(* CoDeSys 2.3 library: beckhoff_network_112.lib *)
(* Libraries: oscat.lib 2.2.11 20:48:25, TcBase.lib 14.5.09 13:14:08, TcSystem.lib 9.3.10 12:21:30, TcpIp.lib 29.5.06 10:26:36, Standard.lib 5.6.98 13:03:02 *)

(* Global variable list: Constants *)
(* @OBJECTFLAGS := '0, 8' *)
VAR_GLOBAL CONSTANT
	NETWORK_BUFFER_LONG_SIZE : UINT := 3999;
	NETWORK_BUFFER_SHORT_SIZE : UINT := 1459;
	LOG_MAX : INT := 40;
	LOG_SIZE : INT := 80;
	ELEMENT_LENGTH : INT := 250;
END_VAR

(* Global variable list: Globale_Variablen *)
VAR_GLOBAL
	TCP_SERVER_RESET : BYTE; (* nur für TwinCAT notwendig ! *)
	LOG_CL : LOG_CONTROL;
END_VAR

(* Data type *)
TYPE DLOG_DATA :
STRUCT
	ADD_HEADER : BOOL;
	ADD_DATA : BOOL;
	CLOCK_TRIG : BOOL;
	ID_MAX : USINT;
	DTI : DT;
	UCB : UNI_CIRCULAR_BUFFER_DATA;
	NEW_FILE : STRING;
	NEW_FILE_RTRIG : BOOL;
END_STRUCT
END_TYPE

(* revision history
ks	01. oct. 2010	rev 1.0
	original version
*)

(* Data type *)
TYPE FILE_PATH_DATA :
STRUCT
	DRIVE : STRING(3);
	DIRECTORY : STRING(STRING_LENGTH);
	FILENAME : STRING;
END_STRUCT
END_TYPE

(* revision history
ks	01. oct. 2010	rev 1.0
	original version
*)

(* Data type *)
TYPE FILE_SERVER_DATA :
STRUCT
	FILE_OPEN : BOOL;
	FILENAME : STRING;
	MODE : BYTE;
	OFFSET : UDINT;
	FILE_SIZE : UDINT;
	AUTO_CLOSE : TIME;
	ERROR : BYTE;
END_STRUCT
END_TYPE

(* revision history
ks	01. oct. 2010	rev 1.0
	original version
*)

(* Data type *)
TYPE IP_C :
STRUCT
	C_MODE : BYTE;						(*W Mode: TCP/UCP AKTIV/PASSIV                               *)
	C_PORT : WORD;						(*W Portnummer                                               *)
	C_IP : DWORD;						(*W IP-Adresse gepackt wwxxyyzz = www.xxx.yyy.zzz            *)
	C_STATE : BYTE;						(*R Verbindungsstatus ON/OFF + Flanke ON/OFF                 *)
	C_ENABLE : BOOL;					(*W Freigabe für Connect                                     *)
	R_OBSERVE : BOOL;					(*W Empfang ueberwachen                                      *)
	TIME_RESET : BOOL;					(*W Alle Timer ruecksetzen                                   *)
	ERROR : DWORD;					(*R vvwwxxyy (vv = CON_ERROR, ww = SEN_ERROR, xx = REC_ERROR *)
	FIFO : IP_FIFO_DATA;					(*I IP FIFO Struktur                                         *)
	MAILBOX : ARRAY [1..16] OF BYTE;	(*I Mailbox: Datenbereich für Bausteindatenaustausch         *)
END_STRUCT
END_TYPE

(* revision history
ks	18. oct. 2008	rev 1.0
	original version
*)

(* Data type *)
TYPE IP_FIFO_DATA :
STRUCT
	X : ARRAY [1..128] OF BYTE; 	(* IP_ID FIFO Speicher          *)
	Y : ARRAY [1..128] OF BYTE; 	(* IP_ID Zähler                 *)
	ID : BYTE;					(* höchste vergabene id         *)
	MAX_ID : BYTE;				(* maximal Anmeldungen pro ID   *)
	INIT : BOOL;					(* Initialisierung durchgeführt *)
	EMPTY : BOOL;				(* FIFO leer                    *)
	FULL : BOOL;					(* FIFO voll                    *)
	TOP : INT;					(* maximale anzahl in FIFO      *)
	NW : INT;					(* Schreibzeiger                *)
	NR : INT;						(* Lesezeiger                   *)
END_STRUCT
END_TYPE

(* revision history
ks	18. oct. 2008	rev 1.0
	original version
*)

(* Data type *)
TYPE IP2GEO_DATA :
STRUCT
	STATE : BOOL;
	IP4 : DWORD;
	COUNTRY_CODE : STRING(2);
	COUNTRY_NAME : STRING(20);
	REGION_CODE : STRING(2);
	REGION_NAME : STRING(20);
	CITY : STRING(20);
	GEO_LATITUDE : REAL;
	GEO_LONGITUDE : REAL;
	TIME_ZONE_NAME : STRING(20);
	GMT_OFFSET : INT;
	IS_DST : BOOL;
END_STRUCT
END_TYPE

(* revision history
ks	14. aug. 2009	rev 1.0
	original version
*)

(* Data type *)
TYPE LOG_CONTROL :
STRUCT
	NEW_MSG : STRING(LOG_SIZE); (* neue Nachricht für den Datenbuffer *)
	NEW_MSG_OPTION : DWORD;
	LEVEL : BYTE;
	SIZE : INT := LOG_MAX; (* Anzahl der Strings im LOG_DATA *)
	RESET : BOOL; (* Nachrichtenbuffer löschen *)
	ENABLE : BOOL := TRUE; (* Debug Logging aktiv *)
	PRINTF : PRINTF_DATA; (* Array PRINTF Parameter *)
	MSG : ARRAY [0..LOG_MAX] OF STRING(LOG_SIZE); (* Array Message *)
	MSG_OPTION : ARRAY [0..LOG_MAX] OF DWORD; (* Array Options *)
	UPDATE_COUNT : UINT; (* Updatezähler *)
	IDX : INT; (* aktueller Nachrichten-Index *)
	RING_MODE : BOOL; (* Bufferüberlauf erkannt *)
END_STRUCT
END_TYPE

(* revision history
ks	18. oct. 2008	rev 1.0
	original version
*)

(* Data type *)
TYPE NETWORK_BUFFER :
STRUCT
	SIZE : UINT;
	BUFFER : NW_BUF_LONG;
END_STRUCT
END_TYPE

(* revision history
ks	01. 01. 2009	rev 1.0
	original version
*)

(* Data type *)
TYPE NETWORK_BUFFER_SHORT :
STRUCT
	SIZE : UINT;
	BUFFER : NW_BUF_SHORT;
END_STRUCT
END_TYPE

(* revision history
ks	01. 01. 2009	rev 1.0
	original version
*)

(* Data type *)
TYPE
	NW_BUF_LONG  : ARRAY[0..NETWORK_BUFFER_LONG_SIZE] OF BYTE;
END_TYPE

(* revision history
ks	01. 01. 2009	rev 1.0
	original version
*)

(* Data type *)
TYPE
	NW_BUF_SHORT : ARRAY[0..NETWORK_BUFFER_SHORT_SIZE] OF BYTE;
END_TYPE

(* revision history
ks	01. 01. 2009	rev 1.0
	original version
*)

(* Data type *)
TYPE PRINTF_DATA : ARRAY [1..11]  OF STRING(LOG_SIZE);
END_TYPE

(* revision history
ks	18. oct. 2008
	original version
*)

(* Data type *)
TYPE UNI_CIRCULAR_BUFFER_DATA :
STRUCT
	D_MODE : INT;
	D_HEAD : WORD;
	D_STRING : STRING(STRING_LENGTH);
	D_REAL : REAL;
	D_DWORD : DWORD;
	BUF_SIZE : UINT;
	BUF_COUNT : UINT;
	BUF_USED : USINT;
	BUF : NW_BUF_LONG;
	_GetStart : UINT;
	_GetEnd : UINT;
	_Last : UINT;
	_First : UINT;
END_STRUCT
END_TYPE

(* revision history
ks	01. oct. 2010	rev 1.0
	original version
*)

(* Data type *)
TYPE URL :
STRUCT
	PROTOCOL : STRING(10);
	USER : STRING(32);
	PASSWORD : STRING(32);
	DOMAIN : STRING(80);
	PORT : WORD;
	PATH : STRING(80);
	QUERY : STRING(STRING_LENGTH);
	ANCHOR : STRING(40);
	HEADER : STRING(160);
END_STRUCT
END_TYPE

(* revision history
hm	18. oct. 2008 v1.0
	original version

ks	01.oct.2010 v1.1
	new header element and string size
*)

(* Data type *)
TYPE us_LOG_VIEWPORT :
STRUCT
	LINE_ARRAY : ARRAY [1..40] OF INT;
	COUNT : INT; (* Anzahl der sichtbaren Nachtrichten *)
	UPDATE_COUNT : UINT; (* Updatezähler *)
	MOVE_TO_X : INT; (* Steuerung der Nachrichtenanzeige *)
	UPDATE : BOOL; (* Daten wurden geändert -> neuzeichnen *)
END_STRUCT
END_TYPE

(* revision history
ks	18. oct. 2008	rev 1.0
	original version
*)

(* Data type *)
TYPE us_TN_INPUT_CONTROL :
STRUCT
	bo_Enable: BOOL; (* Bearbeitung freigeben/sperren *)
	bo_Update_all: BOOL; (* All Elemente neu zeichnen *)
	bo_Reset_Fokus: BOOL; (* Fokus auf 1. Element setzen *)
	in_Focus_at: INT; (* Controlelement mit aktivem Fokus *)
	in_Count: INT; (* Anzahl der benutzen Control-Elemente *)
	in_ToolTip_X: INT; (* Tooltip Text X-Offset *)
	in_ToolTip_Y: INT; (* Tooltip Text Y-Offset *)
	by_ToolTip_Attr: BYTE; (* Tooltip Text Attribute *)
	in_ToolTip_Size: INT; (* Tooltip Text länge *)
	usa_TN_INPUT_CONTROL_DATA: ARRAY [1..20] OF us_TN_INPUT_CONTROL_DATA;
END_STRUCT
END_TYPE

(* revision history
ks	12. mai 2010	rev 1.0
	original version

*)

(* Data type *)
TYPE us_TN_INPUT_CONTROL_DATA :
STRUCT
 	by_Input_Exten_Code: BYTE;
	by_Input_ASCII_Code: BYTE;
	bo_Input_ASCII_IsNum: BOOL;
	in_Title_X_Offset: INT; (* Title Text X-Offset *)
	in_Title_Y_Offset: INT; (* Title Text Y-Offset *)
	by_Title_Attr: BYTE; (* Title Text Attribute *)
	st_Title_String: STRING; (* Title Text String *)
	in_Cursor_X: INT; (* aktuelle Cursor X-Position *)
	in_Cursor_Y: INT; (* aktuelle Cursor Y-Position *)
	in_Type: INT; (* Type des Elements *)
	in_X: INT; (* Element X-Position *)
	in_Y: INT; (* Element Y-Position *)
	in_Cursor_Pos: INT; (* aktuelle Cursorposition *)
	by_Attr_mF: BYTE; (* Text Attribute mit Fokus *)
	by_Attr_oF: BYTE; (* Text Attribute ohne Fokus *)
	in_selected: INT; (* Text Item wurde ausgewählt *)
	st_Input_Mask: STRING; (* Text Eingabemaske *)
	st_Input_Data: STRING(STRING_LENGTH); (* Text aktuelle Eingabedaten *)
	st_Input_String: STRING; (* Text Kopie nach Return-Taste *)
	st_Input_ToolTip: STRING; (* Text ToolTip (Eingabeinformation) *)
	in_Input_Option: INT; (* Text Ausgabe-Optionen *)
	bo_Input_Entered: BOOL; (* RETURN-Taste wurde betätigt *)
	bo_Input_Hidden: BOOL; (* Text versteckete Eingabe mit '*' *)
	bo_Input_Only_Num: BOOL; (* Text nur Nummerneingabe zulassen *)
	bo_Focus: BOOL; (* Element besitzt den Fokus *)
	bo_Update_Input: BOOL; (* Element wegen Benutzereingabe neuzeichnen *)
	bo_Update_All: BOOL; (* Element komplett neuzeichnen *)

END_STRUCT
END_TYPE

(* revision history
ks	12. mai 2010	rev 1.0
	original version

*)

(* Data type *)
TYPE us_TN_MENU :
STRUCT
	st_Menu_Text: STRING(STRING_LENGTH); (* X Menue Texte *)
	in_Menu_E_Count: INT; (* Menue Elemente Anzahl *)
	in_Y: INT; (* Menue Zeilennummer  Y-Position *)
	in_X: INT; (* Menue Spaltennummer X-Position *)
	by_Attr_mF: BYTE; (* Text Attribute mit Fokus *)
	by_Attr_oF: BYTE; (* Text Attribute ohne Fokus *)
	in_X_SM_new: INT; (* neue Sub-Menu X-Position *)
	in_Y_SM_new: INT; (* neue Sub-Menu Y-Position *)
	in_X_SM_old: INT; (* alte Sub-Menu X-Position *)
	in_Y_SM_old: INT; (* alte Sub-Menu Y-Position *)
	in_Cur_Menu_Item: INT; (* aktuelles Haupt-Menue *)
	in_Cur_Sub_Item: INT; (* aktuelles Sub-Menue *)
	in_State: INT; (*   Menu status   *)
	in_Menu_Selected: INT; (* X Menu-Item mit Enter angewwählt *)
	bo_Create: BOOL; (* X Menu erzeugen *)
	bo_Destroy: BOOL; (* X Menu entfernen *)
	bo_Update: BOOL; (* X Menu updaten *)
END_STRUCT
END_TYPE

(* revision history
ks	12. mai 2010	rev 1.0
	original version

*)

(* Data type *)
TYPE us_TN_MENU_POPUP :
STRUCT
	st_Menu_Text: STRING(STRING_LENGTH); (* X Menue Texte *)
	in_Menu_E_Count: INT; (* Menue Elemente Anzahl *)
	in_X: INT; (* X Menue X-Position *)
	in_Y: INT; (* X Menue Y-Position *)
	in_Cols: INT; (* Menue Spaltenanzahl *)
	in_Rows: INT; (* Menue Zeilenanzahl *)
	in_Cur_Item: INT; (* X aktuelles Sub-Menue *)
	by_Attr_mF: BYTE; (* X Text Attribute mit Fokus	*)
	by_Attr_oF: BYTE; (* X Text Attribute ohne Fokus *)
	by_Input_Exten_Code: BYTE; (* X Tastencode: Sondertasten *)
	bo_Create: BOOL; (* X Popup-Menu erzeugen *)
	bo_Destroy: BOOL; (* X Popup-Menu entfernen *)
	bo_Update: BOOL; (* X Popup-Menu updaten *)
	bo_Activ: BOOL; (*   Popup-Menu ist aktiv *)
END_STRUCT
END_TYPE

(* revision history
ks	12. mai 2010	rev 1.0
	original version

*)

(* Data type *)
TYPE us_TN_SCREEN :
STRUCT
	bya_CHAR: ARRAY [0..1919] OF BYTE;
	bya_COLOR: ARRAY [0..1919] OF BYTE;
	bya_BACKUP: ARRAY [0..1919] OF BYTE;
	bya_Line_Update: ARRAY [0..23] OF BOOL;
	by_Input_Exten_Code: BYTE;
	by_Input_ASCII_Code: BYTE;
	bo_Input_ASCII_IsNum: BOOL;
	in_Page_Number: INT; (* aktive Seiten-Nr. *)
	in_Cursor_X: INT; (* Cursor X-Position *)
	in_Cursor_Y: INT; (* Cursor Y-Position *)
	in_EOS_Offset: INT; (* End of String Offset *)
	by_Clear_Screen_Attr: BYTE; (* Clear-Screen Attr *)
	bo_Clear_Screen: BOOL; (* Clear-Screen auslösen *)
	bo_Modal_Dialog: BOOL; (* Modaler Dialog ist aktiv *)
	bo_Menue_Bar_Dialog: BOOL; (* Menue Dialog ist aktiv *)
END_STRUCT
END_TYPE

(* revision history
ks	12. mai 2010	rev 1.0
	original version

*)

(* Data type *)
TYPE VMAP_DATA :
STRUCT
	FC : DWORD;
	V_ADR : INT;
	V_SIZE : INT;
	P_ADR : INT;
	TIME_OUT : TIME;
END_STRUCT
END_TYPE

(* revision history
ks	18. oct. 2008	rev 1.0
	original version
*)

(* Data type *)
TYPE WORLD_WEATHER_CUR :
STRUCT
	OBSERVATION_TIME : STRING(8);
	TEMP_C : INT;
	WEATHER_CODE : INT;
	WEATHER_DESC : STRING(30);
	WIND_SPEED_MILES : INT;
	WIND_SPEED_KMPH : INT;
	WIND_DIR_DEGREE : INT;
	WIND_DIR16POINT : STRING(3);
	PRECIPMM : REAL;
	HUMIDITY : INT;
	VISIBILITY : INT;
	PRESSURE : INT;
	CLOUDOVER : INT;
END_STRUCT
END_TYPE

(* revision history
ks	01. oct. 2010	rev 1.0
	original version

*)

(* Data type *)
TYPE WORLD_WEATHER_DATA :
STRUCT
	CUR : WORLD_WEATHER_CUR;
	DAY : ARRAY [0..4] OF WORLD_WEATHER_DAY;
END_STRUCT
END_TYPE

(* revision history
ks	01. oct. 2010	rev 1.0
	original version

*)

(* Data type *)
TYPE WORLD_WEATHER_DAY :
STRUCT
	DATE_OF_DAY : STRING(10);
	TEMP_MAX_C : INT;
	TEMP_MAX_F : INT;
	TEMP_MIN_C : INT;
	TEMP_MIN_F : INT;
	WIND_SPEED_MILES : INT;
	WIND_SPEED_KMPH : INT;
	WIND_DIR_DEGREE : INT;
	WIND_DIR16POINT : STRING(3);
	WEATHER_CODE : INT;
	WEATHER_DESC : STRING(30);
	PRECIPMM : REAL;
END_STRUCT
END_TYPE

(* revision history
ks	01. oct. 2010	rev 1.0
	original version

*)

(* Data type *)
TYPE XML_CONTROL :
STRUCT
	COMMAND : WORD;
	WATCHDOG : TIME;
	START_POS : UINT;
	STOP_POS : UINT;
	COUNT : UINT;
	TYP : INT;
	LEVEL : UINT;
	PATH : STRING(STRING_LENGTH);
	ELEMENT : STRING(STRING_LENGTH);
	ATTRIBUTE : STRING(STRING_LENGTH);
	VALUE : STRING(STRING_LENGTH);
	BLOCK1_START : UINT;
	BLOCK1_STOP : UINT;
	BLOCK2_START : UINT;
	BLOCK2_STOP : UINT;
END_STRUCT
END_TYPE

(* revision history
ks	18. oct. 2008	rev 1.0
	original version

ks	24. sep. 2010	rev 1.1
	STRING(STRING_LENGTH)
*)

(* Data type *)
TYPE YAHOO_WEATHER_DATA :
STRUCT
	TIMETOLIVE : INT;							(* TIME TO LIVE: HOW LONG IN MINUTES THIS FEED SHOULD BE CACHED         *)
	LOCATION_CITY : STRING(40);   				(* THE LOCATION OF THIS FORECAST: CITY: CITY NAME  *)
	LOCATION_REGION : STRING(20);  				(* THE LOCATION OF THIS FORECAST: REGION: STATE, TERRITORY, OR REGION, IF GIVEN *)
	LOCATION_COUNTRY : STRING(20);			(* THE LOCATION OF THIS FORECAST: COUNTRY: TWO-CHARACTER COUNTRY CODE *)
	UNIT_TEMPERATURE : STRING(1);				(* TEMPERATURE: DEGREE UNITS, F FOR FAHRENHEIT OR C FOR CELSIUS *)
	UNIT_DISTANCE : STRING(2);					(* DISTANCE: UNITS FOR DISTANCE, MI FOR MILES OR KM FOR KILOMETERS *)
	UNIT_PRESSURE : STRING(2);					(* PRESSURE: UNITS OF BAROMETRIC PRESSURE, IN FOR POUNDS PER SQUARE INCH OR MB FOR MILLIBARS *)
	UNIT_SPEED : STRING(4);						(* SPEED: UNITS OF SPEED, MPH FOR MILES PER HOUR OR KPH FOR KILOMETERS PER HOUR *)
	WIND_CHILL : INT;							(* FORECAST INFORMATION ABOUT WIND CHILL IN DEGREES *)
	WIND_DIRECTION : INT;						(* FORECAST INFORMATION ABOUT WIND DIRECTION, IN DEGREES *)
	WIND_SPEED : REAL;							(* FORECAST INFORMATION ABOUT WIND SPEED, IN THE UNITS (MPH OR KPH)*)
	ATMOSPHERE_HUMIDITY : INT;				(* FORECAST INFORMATION ABOUT CURRENT ATMOSPHERIC HUMIDITY: HUMIDITY, IN PERCENT  *)
	ATMOSPHERE_PRESSURE : INT;				(* FORECAST INFORMATION ABOUT CURRENT ATMOSPHERIC PRESSURE: BAROMETRIC PRESSURE, IN THE UNITS (IN OR MB) *)
	ATMOSPHERE_VISIBILITY : REAL;				(* FORECAST INFORMATION ABOUT CURRENT ATMOSPHERIC VISIBILITY, IN THE UNITS (MI OR KM) *)
	ATMOSPHERE_RISING : INT;					(* FORECAST INFORMATION ABOUT RISING: STATE OF THE BAROMETRIC PRESSURE: STEADY (0), RISING (1), OR FALLING (2). (INTEGER: 0, 1, 2) *)
	ASTRONOMY_SUNRISE : STRING(10);			(* SUNRISE: TODAY'S SUNRISE TIME. THE TIME IS A STRING IN A LOCAL TIME FORMAT OF "H:MM AM/PM" *)
	ASTRONOMY_SUNSET : STRING(10);			(* SUNSET: TODAY'S SUNSET TIME. THE TIME IS A STRING IN A LOCAL TIME FORMAT OF "H:MM AM/PM", *)
	GEO_LATITUDE : REAL;						(* THE LATITUDE OF THE LOCATION *)
	GEO_LONGITUDE : REAL;						(* THE LONGITUDE OF THE LOCATION *)
	CUR_CONDITIONS_TEMP : INT;				(* THE CURRENT WEATHER CONDITIONS: TEMP: THE CURRENT TEMPERATURE, IN THE UNITS (F OR C) *)
	CUR_CONDITIONS_TEXT : STRING(40);			(* THE CURRENT WEATHER CONDITIONS: TEXT: A TEXTUAL DESCRIPTION OF CONDITIONS *)
	CUR_CONDITIONS_CODE : INT;				(* THE CURRENT WEATHER CONDITIONS: CODE: THE CONDITION CODE FOR THIS FORECAST *)
	FORCAST_TODAY_LOW_TEMP : INT;			(* THE FORCAST TODAY WEATHER CONDITIONS: THE FORECASTED LOW TEMPERATURE FOR THIS DAY IN THE UNITS (F OR C) *)
	FORCAST_TODAY_HIGH_TEMP : INT;			(* THE FORCAST TODAY WEATHER CONDITIONS: THE FORECASTED HIGH TEMPERATURE FOR THIS DAY IN THE UNITS (F OR C) *)
	FORCAST_TODAY_TEXT : STRING(40);			(* THE FORCAST TODAY WEATHER CONDITIONS: TEXT: A TEXTUAL DESCRIPTION OF CONDITIONS *)
	FORCAST_TODAY_CODE : INT;				(* THE CURRENT WEATHER CONDITIONS: CODE: THE CONDITION CODE FOR THIS FORECAST *)
	FORCAST_TOMORROW_LOW_TEMP : INT; 		(* THE FORCAST TOMORROW WEATHER CONDITIONS: THE FORECASTED LOW TEMPERATURE FOR THIS DAY IN THE UNITS (F OR C) *)
	FORCAST_TOMORROW_HIGH_TEMP : INT;		(* THE FORCAST TOMORROW WEATHER CONDITIONS: THE FORECASTED HIGH TEMPERATURE FOR THIS DAY IN THE UNITS (F OR C) *)
	FORCAST_TOMORROW_TEXT : STRING(40);	(* THE FORCAST TOMORROW WEATHER CONDITIONS: TEXT: A TEXTUAL DESCRIPTION OF CONDITIONS *)
	FORCAST_TOMORROW_CODE : INT;			(* THE CURRENT WEATHER CONDITIONS: CODE: THE CONDITION CODE FOR THIS FORECAST *)

END_STRUCT
END_TYPE

(* revision history
ks	18. oct. 2008	rev 1.0
	original version

ks	24. sep. 2010	rev 1.1
	LOCATION_COUNTRY STRING(20)

*)

(* POU BASE64_DEMO, CFC *)
PROGRAM BASE64_DEMO
VAR
	text1: STRING(144) := '<4036.1076324381@guildenstern.zeitform.de>';
	text2: STRING(192);
	text3: STRING(144);
	BASE64_DECODE_STR: BASE64_DECODE_STR;
	BASE64_ENCODE_STR: BASE64_ENCODE_STR;
	start: BOOL := TRUE;
	done1: BOOL;
	done2: BOOL;
END_VAR
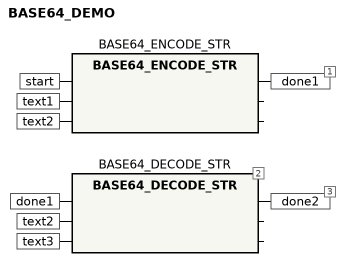
_CFC_ (* Continuous Function Chart, elements in execution order *)
#0 BASE64_ENCODE_STR:BASE64_ENCODE_STR(start, text1, text2)
#1 done1 <= #0.out 1
#2 BASE64_DECODE_STR:BASE64_DECODE_STR(done1, text2, text3)
#3 done2 <= #2.out 1
_END_CFC_
END_PROGRAM

(* POU BASE64_DECODE_STR, ST *)
FUNCTION_BLOCK BASE64_DECODE_STR
VAR_INPUT
	RUN : BOOL;
END_VAR
VAR_OUTPUT
	DONE : BOOL;
END_VAR
VAR_IN_OUT
	STR1 : STRING(192);
	STR2 : STRING(144);
END_VAR
VAR
	BASE64_DECODE_STREAM : BASE64_DECODE_STREAM;
	run_last : BOOL;
	buf1 : ARRAY [0..63] OF BYTE;
	buf2 : ARRAY [0..47] OF BYTE;
	mode : INT;
	size1 : INT;
	size2 : INT;
	end : INT;
	pos : INT;
END_VAR

(*
version 1.0	06. dec. 2009
programmer 	ks
tested by	ks

BASE64_DECODE_STR konvertiert einen BASE64 kodierten String in einen normalen String. 

*)
CASE mode OF
0:	IF RUN AND NOT run_last THEN
		DONE := FALSE;
		mode := 1;
		end := LEN(STR1);
		pos := 0;
		STR2 := '';
	END_IF;
1:
	size1 := MIN(48,end - pos);
	IF size1 > 0 THEN
		_STRING_TO_BUFFER(STR:=MID(STR1, size1, pos + 1), POS:=0, PT:=ADR(buf1), SIZE:=SIZEOF(buf1));
		BASE64_DECODE_STREAM(BUF1:=buf1 ,BUF2:=buf2 ,SIZE1:=size1 ,SIZE2=>size2);
		STR2 := CONCAT(STR2,BUFFER_TO_STRING(PT:=ADR(buf2), SIZE:=SIZEOF(buf2), START:=0, STOP:=size2 - 1));
	ELSE
		mode := 0;
		DONE := TRUE;
	END_IF;
	pos := pos + size1;
END_CASE;

run_last := RUN;

(* revision history

ks	6. dec. 2009 rev 1.0
	original version

*)
END_FUNCTION_BLOCK

(* POU BASE64_DECODE_STREAM, ST *)
FUNCTION_BLOCK BASE64_DECODE_STREAM
VAR_IN_OUT
	BUF1 : ARRAY [0..63] OF BYTE;
	BUF2 : ARRAY [0..47] OF BYTE;
END_VAR
VAR_INPUT
	SIZE1 : INT;
END_VAR
VAR_OUTPUT
	SIZE2 : INT;
END_VAR
VAR_TEMP
	a: INT;
	b: WORD;
	o: INT;
	off: INT;
	i1: INT;
	i2: INT;
	c: INT;
END_VAR

(*
version 1.0	06. dec. 2009
programmer 	ks
tested by	ks

BASE64_DECODE_STREAM konvertiert einzelne Base64 kodierte Datenblöcke in normalen Datenblöcke. 

*)
IF SIZE1 <= 0 THEN SIZE2 := 0; RETURN; END_IF;
c := SIZE1 - 1;
i2 := 0;
a := 0;
b := 0;
FOR i1 := 0 TO c DO
	o := BUF1[i1];
	IF o = 61  (* = *) THEN	EXIT;
	ELSIF o > 96 (* a-z *) THEN off := 71;
	ELSIF o > 64 (* A-Z *) THEN off := 65;
	ELSIF o > 47 (* 0-9 *) THEN off := -4;
	ELSIF o = 43 (* + *) THEN off := -19;
	ELSIF o = 47 (* / *) THEN off := -16;
	END_IF;
	b := SHL(b,6) OR INT_TO_BYTE(o - off);
	a := a + 6;
	IF a >= 8 THEN
		a := a - 8;
		BUF2[i2] := WORD_TO_BYTE(SHR(b,a));
		i2 := i2 + 1;
		b := b AND NOT SHL(WORD#16#FFFF,a);
	END_IF;
END_FOR;
SIZE2 := i2;

(* revision history

ks	6. dec. 2009 rev 1.0
	original version

*)
END_FUNCTION_BLOCK

(* POU BASE64_ENCODE_STR, ST *)
FUNCTION_BLOCK BASE64_ENCODE_STR
VAR_INPUT
	RUN : BOOL;
END_VAR
VAR_OUTPUT
	DONE : BOOL;
END_VAR
VAR_IN_OUT
	STR1 : STRING(144);
	STR2 : STRING(192);
END_VAR
VAR
	BASE64_ENCODE_STREAM : BASE64_ENCODE_STREAM;
	run_last : BOOL;
	buf1 : ARRAY [0..47] OF BYTE;
	buf2 : ARRAY [0..63] OF BYTE;
	mode : INT;
	size1 : INT;
	size2 : INT;
	end : INT;
	pos : INT;
END_VAR

(*
version 1.0	06. dec. 2009
programmer 	ks
tested by	ks

BASE64_ENCODE_STR konvertiert einen normalen String in einen BASE64 kodierten String. 

*)
CASE mode OF
0:	IF RUN AND NOT run_last THEN
		DONE := FALSE;
		mode := 1;
		end := LEN(STR1);
		pos := 0;
		STR2 := '';
	END_IF;
1:
	size1 := MIN(48,end - pos);
	IF size1 > 0 THEN
		_STRING_TO_BUFFER(STR:=MID(STR1, size1, pos + 1), POS:=0, PT:=ADR(buf1), SIZE:=SIZEOF(buf1));
		BASE64_ENCODE_STREAM(BUF1:=buf1 ,BUF2:=buf2 ,SIZE1:=size1 ,SIZE2=>size2);
		STR2 := CONCAT(STR2,BUFFER_TO_STRING(PT:=ADR(buf2), SIZE:=SIZEOF(buf2), START:=0, STOP:=size2 - 1));
	ELSE
		mode := 0;
		DONE := TRUE;
	END_IF;
	pos := pos + size1;
END_CASE;

run_last := RUN;

(* revision history

ks	6. dec. 2009 rev 1.0
	original version

*)
END_FUNCTION_BLOCK

(* POU BASE64_ENCODE_STREAM, ST *)
FUNCTION_BLOCK BASE64_ENCODE_STREAM
VAR_IN_OUT
	BUF1 : ARRAY [0..47] OF BYTE;
	BUF2 : ARRAY [0..63] OF BYTE;
END_VAR
VAR_INPUT
	SIZE1 : INT;
END_VAR
VAR_OUTPUT
	SIZE2 : INT;
END_VAR
VAR
	a: INT;
	b: WORD;
	i: INT;
	i2: INT;
	i3: INT;
	c: INT;
	BASE64: STRING(64) := 'ABCDEFGHIJKLMNOPQRSTUVWXYZabcdefghijklmnopqrstuvwxyz0123456789+/';
END_VAR

(*
version 1.0	06. dec. 2009
programmer 	ks
tested by	ks

BASE64_ENCODE_STREAM konvertiert Datenblöcke in Base64. 

*)
IF SIZE1 <= 0 THEN
	SIZE2 := 0;
	RETURN;
END_IF;
c := SIZE1 - 1;
i2 := 0;
a := 0;
b := 0;
FOR i := 0 TO c DO
	b := SHL(b,8) OR BUF1[i];
	a := a + 8;
	WHILE a >= 6 DO
		a := a - 6;
		buf2[i2] := CODE(BASE64,WORD_TO_INT(SHR(b,a)) + 1);
		i2 := i2 + 1;
		b := b AND NOT SHL(WORD#16#FFFF,a);
	END_WHILE;
END_FOR;
IF a > 0 THEN
	buf2[i2] := CODE(BASE64,WORD_TO_INT(SHL(b,6 - a)) + 1);
	i2 := i2 + 1;
	i3 := i2 + (NOT INT_TO_WORD(i2) AND 2#11);
	FOR i := i2 TO i3 DO
		buf2[i] := 61;
	END_FOR;
	SIZE2 := i3 + 1;
ELSE
	SIZE2 := i2;
END_IF;

(* revision history

ks	6. dec. 2009 rev 1.0
	original version

*)
END_FUNCTION_BLOCK

(* POU CSV_PARSER_BUF_DEMO, ST *)
PROGRAM CSV_PARSER_BUF_DEMO
VAR CONSTANT
	 line_cnt : INT:=2;
	 col_cnt : INT:=4;
END_VAR
VAR
	CPB : CSV_PARSER_BUF;
	FS : FILE_SERVER;
	FSD : FILE_SERVER_DATA;
	PT : NETWORK_BUFFER;
	sep : BYTE;
	value : STRING(STRING_LENGTH);
	step : INT;
	result : BYTE;
	offset : UDINT;
	run : BYTE;
	done : BOOL;
	value_real : REAL;
	cnt : INT;
	line : INT;
	idx : INT;
	data : ARRAY [1..line_cnt, 1..col_cnt] OF REAL;
	FB_LOG_MESSAGE : LOG_MSG;
END_VAR
(* Demo-Programm: CSV-Datei mittels Enumeration auswerten
die groesse des arrays kann mittels konstanten line_cnt und col_cnt angepasst werden

 ----- den nachfolgenden Textblock als datei "csv.txt" auf der sps ablegen ---
10.45,20,30,40.8
115,3450.2123,456,123.1
---------------------------------------------------------------------------------*)

CASE step OF

00:	IF NOT done THEN
	 	(* File_Daten einrichten  *)
		FSD.FILENAME := 'd:\pxc\oscat\network\csv.txt'; (* Dateiname *)
		FSD.MODE := 1; (* vorhandene Datei zum lesen öffnen *)
		FSD.OFFSET := 0; (* Start bei Dateianfang *)
		FSD.AUTO_CLOSE := T#0s; (* kein Auto-Close verwenden *)
		PT.SIZE := 65535; (* maximale länge einlesen *)
		step := 10;
	END_IF;

10:	IF FSD.MODE = 0 THEN (* Datei geöffnet ? *)
		OFFSET := 0; (* Start Offset vorgeben *)
		sep :=44; (* Trennzeichen , *)
		run := 1; (* Element suchen *)
		cnt := 0;
		step := 20;
	END_IF;

20:	IF run = 0 THEN
		(* ---------------------- Debug-Message ----------------------------*)
		IF LOG_CL.ENABLE THEN
			LOG_CL.NEW_MSG := 'CPFD: /value >~2< /offset ~3 /Run ~4 /Result ~5';
			LOG_CL.PRINTF[2] := value;
			LOG_CL.PRINTF[3] := UDINT_TO_STRING(OFFSET);
			LOG_CL.PRINTF[4] := BYTE_TO_STRING(run);
			LOG_CL.PRINTF[5] := BYTE_TO_STRING(result);
			FB_LOG_MESSAGE();
		END_IF;
		(* -----------------------------------------------------------------*)

		run := 1; (*  nächstes Element suchen  *)

		IF result = 1 OR result = 2 THEN
			(* automatische konvertierung in real ausführen *)
			IF LEN(value) <= 20 THEN
				value_real := FLOAT_TO_REAL(FLT:=value);
			ELSE
				value_real := 0.0;
			END_IF;

			cnt := cnt + 1;
			IF cnt <= line_cnt * col_cnt THEN
				line := (cnt / col_cnt) + 1;
				idx := (cnt MOD col_cnt);
				data[line,idx] := value_real; (* Daten in Array eintragen *)
			END_IF;

		ELSIF result = 10 THEN (* nichts mehr gefunden *)
			run := 0; (* keine weitere INI Auswertung erwünscht *)
			FSD.MODE := 5; (* Datei schliessen *)
			step := 30;
		END_IF;
	END_IF;

30:	IF FSD.MODE = 0 THEN (* Datei geschlossen ? *)
		step := 0;
		done := TRUE;
	END_IF;

END_CASE;

CPB(SEP:=sep,RUN:=run,OFFSET:=OFFSET,VALUE:=value,PT:=PT,RESULT=>result); (* CSV PARAMETER BUF *)
FS(FSD:=FSD,PT:=PT); (* FILE_SERVER *)
END_PROGRAM

(* POU CSV_PARSER_BUF, ST *)
FUNCTION_BLOCK CSV_PARSER_BUF
VAR_INPUT
	SEP : BYTE;
END_VAR
VAR_IN_OUT
	RUN : BYTE;
	OFFSET : UDINT;
	VALUE : STRING(STRING_LENGTH);
	PT : NETWORK_BUFFER;
END_VAR
VAR_OUTPUT
	RESULT : BYTE;
END_VAR
VAR
	step : INT;
	size : INT;
	c : BYTE;
	v_add : BYTE;
	i : INT;
	state : BYTE;
	eof : BOOL;
	pv : POINTER TO BYTE;
	pve : DWORD;
	watchdog : TON;
	x : BOOL;

	(*FB_LOG_MESSAGE : LOG_MSG;
	_debug_enable : BOOL := TRUE;
	step_last : INT;*)
END_VAR

(*
version 1.0		01. oct. 2010
programmer 		ks
tested by			ks

CSV_PARSER_BUF liefert die Elemente oder Zeilen einer Textdatei die in einem Bytearray abgelegt ist.

--------------------------------------

RUN Mode
00 = kein Befehl aktiv
01 = Element suchen

Result Codes
01 = Element gefunden
02 = Element und Zeilenende erkannt
05 = Befehl in Arbeit (Busy)
10 = nichts gefunden - Daten-Ende erreicht

State Codes
01 = Element gefunden
02 = Element und Zeilenende erkannt
05 = Befehl in Arbeit (Busy)
10 = nichts gefunden - Daten-Ende erreicht

*)
IF RUN > 0 THEN
	IF state = 0 THEN (* Auswertung neu beginnen *)

		pv := ADR(VALUE);
		pv^ := 0; (* VALUE = '' *)
		pve := pv + INT_TO_DWORD(STRING_LENGTH);
		i := UDINT_TO_INT(OFFSET);
		size := UINT_TO_INT(PT.SIZE) - 1;
		RESULT := 0;
		state := 5; (* Befehl in Arbeit (Busy) *)
		step := 0; (* Auswertung neu beginnen *)

		(* ---------------- Debug-Message -----------------------*)
		(*IF _debug_enable THEN
			LOG_CL.NEW_MSG := 'CPF: Startindex: ~1';
			LOG_CL.PRINTF[1] := INT_TO_STRING(i);
			FB_LOG_MESSAGE();
		END_IF;*)
		(* -----------------------------------------------------------------*)

	END_IF;

	watchdog(IN:=FALSE,PT:=T#1ms); (* Timer neustarten *)
	watchdog.IN := TRUE;

	WHILE (state = 5) DO (* Schleife solange kein Ergebnis *)

		watchdog(); (* Timer aktualisieren *)

		IF watchdog.Q THEN (* watchdog ausgelöst *)
			state := 5;
			EXIT;
		ELSIF i > size THEN (* kein weiteres zeichen vorhanden *)
			state := 10; (* nichts gefunden - Daten-Ende erreicht *)
			EXIT;
		ELSE

			c := PT.BUFFER[i]; (* neues Zeichen aus Buffer lesen *)
			eof := i + 1 = PT.SIZE; (* End of File *)

			v_add := 0;

			IF c = SEP THEN (* Neues Element erkannt *)
				state := 1;
				x := TRUE;
			ELSIF c >= 32 THEN (* Element erkannt *)
				v_add := c; (* Zeichen ablegen *)
				IF eof THEN
					state := 2; (* Element und Zeilenende erkannt *)
				ELSE
					x := TRUE;
				END_IF;
			ELSE
				IF x THEN
					state := 2; (* Element und Zeilenende erkannt *)
					x := FALSE;
				END_IF;
			END_IF;

			IF v_add > 0  AND pv < pve THEN (* Zeichen zu Value-String hinzufügen *)
				pv^ := v_add; (* Zeichen eintragen *)
				pv := pv + 1;
				pv^ := 0; (* String-Terminierung eintragen *)
			END_IF;

			i := i + 1; (* Datenzeiger erhöhen *)

		END_IF;
	END_WHILE;

	CASE state OF
	01:	(* Element gefunden *)
		RESULT := 1; (* Element gefunden *)
		OFFSET := i; (* Offset uebernehmen *)
		RUN := 0;
		state := 0;
	02:	(* Element gefunden *)
		RESULT := 2; (* Element und Zeilenende erkannt *)
		OFFSET := i; (* Offset uebernehmen *)
		RUN := 0;
		state := 0;

	05:	RESULT := 5; (* in Arbeit *)

	10:	(* Indexüberschreitung - Bufferende *)
		RESULT := 10; (* nichts gefunden - Datenende erreicht *)
		OFFSET := i; (* Offset uebernehmen *)
		RUN := 0;
		state := 0;
	END_CASE;

	(* ---------------- Debug-Message -----------------------*)
	(*IF _debug_enable THEN
		LOG_CL.NEW_MSG := 'CPF: intern Result ~1 , state ~2, step ~3 , offset ~4, run ~5';
		LOG_CL.PRINTF[1] := BYTE_TO_STRING(RESULT);
		LOG_CL.PRINTF[2] := BYTE_TO_STRING(state);
		LOG_CL.PRINTF[3] := INT_TO_STRING(step);
		LOG_CL.PRINTF[4] := UDINT_TO_STRING(OFFSET);
		LOG_CL.PRINTF[5] := BYTE_TO_STRING(RUN);
		FB_LOG_MESSAGE();
	END_IF;*)
	(* -----------------------------------------------------------------*)

END_IF;

(* ---------------- Debug-Message -----------------------*)
(*IF _debug_enable THEN
	IF step_last <> step THEN
		LOG_CL.NEW_MSG := 'IPB: Step: ~1';
		LOG_CL.PRINTF[1]  := INT_TO_STRING(step);
		FB_LOG_MESSAGE();
	END_IF;
	step_last := step;
END_IF;*)
(* -----------------------------------------------------------------*)

(* revision history
ks	01. oct. 2010	rev 1.0
	original version
*)
END_FUNCTION_BLOCK

(* POU FILE_SERVER, ST *)
FUNCTION_BLOCK FILE_SERVER
VAR_IN_OUT
	FSD : FILE_SERVER_DATA;
	PT : NETWORK_BUFFER;
END_VAR
VAR
	buf_size : UDINT;
	handle : UINT; (* Filehandle *)
	read_max_length : UDINT;(* maximale Datenlänge *)
	file_position : UDINT;(* aktueller Schreib/Lesezeiger *)
	used_filename : STRING;(* aktueller Dateiname *)
	close_time : TIME;
	length_read : UDINT;
	write_length : UDINT;
	length_written : UDINT;
	open_handle : UINT;
	seek_position : UDINT;
	seek_mode : INT;
	seek_data : ARRAY[0..1] OF DINT;
	tell_position : UDINT;
	open_mode : DWORD;
	last_mode: BYTE;
	command : BYTE;
	error_code : BYTE;
	error : BOOL;
	file_change : BOOL;
	step : INT;
	t_diff : TIME;
	tx_last : TIME;
	tx : TIME;
	X : FW_AdsRdWrt;
	tmpDW : UDINT;
	para : BOOL;

	(*FB_LOG_MESSAGE : LOG_MSG;
	_debug_enable : BOOL := TRUE;
	step_last : INT;*)
END_VAR

(*
version 1.0		23. sep. 2010
programmer 		ks
tested by			ks

FILE_SERVER ermöglicht den Zugriff auf Datteien mittels Plattform-Neutraler Schnittstelle
*)

(*
- Befehle -
1 = File_Open_Exist + File_Read
2 = File_Open_Exist + File_Write
3 = File_Open_New  + File_Write
4 = File_Remove
5 = File_Close

- Action -
1 = file_open (open)
2 = file_close (close)
3 = file_read (read)
4 = file_write (write)
5 = file_seek (setpos)
6 = file_tell (getpos)
7 = file_remove (delete)

---- fehlermeldungen----

00	Kein Fehler
19	SYSTEMSERVICE_FOPEN		Unbekannte oder ungültige Parameter
28	SYSTEMSERVICE_FOPEN		Datei nicht gefunden. Ungültiger Dateiname oder Dateipfad
38	SYSTEMSERVICE_FOPEN		Keine weiteren freien File Handles.
51	SYSTEMSERVICE_FCLOSE	ungültiges oder unbekanntes file handle.
62	SYSTEMSERVICE_FCLOSE	Datei wurde mit falscher Methode geöffnet.
67	SYSTEMSERVICE_FREAD		ungültiges oder unbekanntes file handle.
74	SYSTEMSERVICE_FREAD		Kein Speicher für Lesebuffer.
78	SYSTEMSERVICE_FREAD		Datei wurde mit falscher Methode geöffnet.
83	SYSTEMSERVICE_FWRITE	ungültiges oder unbekanntes file handle
94	SYSTEMSERVICE_FWRITE	Datei wurde mit falscher Methode geöffnet.
99	SYSTEMSERVICE_FSEEK		ungültiges oder unbekanntes file handle.
110	SYSTEMSERVICE_FSEEK		Datei wurde mit falscher Methode geöffnet.
115	SYSTEMSERVICE_FTELL		ungültiges oder unbekanntes file handle.
126	SYSTEMSERVICE_FTELL		Datei wurde mit falscher Methode geöffnet
140	SYSTEMSERVICE_FDELETE	Datei nicht gefunden. Ungültiger Dateiname oder Dateipfad.
255	Applikation					Position liegt hinter dem Dateiende

*)
(* read system timer *)
tx := UDINT_TO_TIME(T_PLC_MS());
t_diff := tx - tx_last;
tx_last := tx;

CASE step OF
0:
	IF FSD.MODE = LIMIT(1,FSD.MODE,5) THEN

		(* ---------------------- Debug-Message ----------------------------*)
		(*IF _debug_enable THEN
			LOG_CL.NEW_MSG := 'FS: File_Start Mode=~1';
			LOG_CL.PRINTF[1] := BYTE_TO_STRING(FSD.MODE);
			FB_LOG_MESSAGE();
		END_IF;*)
		(* -----------------------------------------------------------------------------*)

		(* Initialisierung *)
		X.sNetId := '';
		X.tTimeout := T#5s;
		X.nPort := 10000; (* AMSPORT_R3_SYSSERV *)

		buf_size := SIZEOF(PT.BUFFER);
		close_time := T#1ms; (* wenn Schritt aktiv ist, dann Close-Timer rücksetzen *)

		IF FSD.MODE = 4 THEN (* File_Remove *)
			IF handle > 0 THEN
				File_change := TRUE;
				step := 32000; (* File_Close ausführen *)
			ELSE
				step := 90; (* File_Remove ausführen *)
			END_IF;

		ELSIF FSD.MODE = 5 THEN (* File_Close *)
			step := 32000; (* File_Close ausführen *)

		ELSIF handle = 0 THEN (* MODE 1,2,3 *)
			step := 100; (* File muss erst geöffnet werden *)

		ELSE (* File ist geöffnset *)
			IF used_filename = FSD.FILENAME AND FSD.MODE = last_mode THEN (* kein Moduswechsel ? *)
				step := 200; (* ohne open prozedure weitermachen *)
			ELSE
				step := 32000;
				File_change := TRUE;
			END_IF;
		END_IF;

	ELSIF handle > 0 THEN (* offene Datei gefunden - AutoClose Modus *)
		IF FSD.AUTO_CLOSE > T#0s THEN
			close_time := close_time + t_diff; (* Close_Time hochzählen *)
			IF close_time > FSD.AUTO_CLOSE THEN (* Zeit überschrittenen *)
				step := 32000; (* automatisch Datei schliessen *)
			END_IF;
		END_IF;
	END_IF;

(* ----------------------------------- *)
090: (* File_Remove *)
	command := 7; (* File Remove *)
	step := 95;

095: (* File_Remove beendet *)
	IF command = 0 THEN
		step := 30000; (* Beenden *)
	END_IF;
(* ----------------------------------- *)

100: (* File_Open *)
	IF FSD.MODE = 3 THEN (* Open_New + File Write *)
		open_mode := 16#0001_001A; (* PATH_GENERIC + WRITEPLUS + BINARY *)
	ELSE (* Mode 1 Open_Exist + File _Read / Mode 2 Open_Exist + File_Write *)
		open_mode := 16#0001_0019; (* PATH_GENERIC + READPLUS + BINARY *)
	END_IF;
	command := 1; (* FileOpen *)
	step := 105;

105: (* File Open beendet *)
	IF command = 0 THEN
		IF error THEN
			step := 30000; (* Beenden *)
		ELSE
			(* Filedaten eintragen *)
			close_time := T#1ms; (* Timer freigeben *)
			handle := open_handle;
			used_filename := FSD.FILENAME;
			file_position := UDINT#4294967295; (* maximal = unbekannt *)
			last_mode := FSD.MODE;
			step := 110;
		END_IF;
	END_IF;

110: (* File Seek *)
	command := 5; (* File-Seek *)
	seek_position := 0;
	seek_mode := 2; (* SEEK_END - Seek from the end of file *)
	step := 115;

115: (* File Seek beendet *)
	IF command = 0 THEN
		IF error THEN
			step := 30000; (* Beenden *)
		ELSE
			command := 6; (* File-Tell starten *)
			step := 120;
		END_IF;
	END_IF;

120: (* File Tell beendet *)
	IF command = 0 THEN
		IF error THEN
			step := 30000; (* Beenden *)
		ELSE
			FSD.FILE_SIZE := tell_position; (* aktuelle Dateigroesse *)
			FSD.FILE_OPEN := TRUE;
			step := 200;
		END_IF;
	END_IF;

200: (* File Seek *)
	IF FSD.OFFSET > FSD.FILE_SIZE THEN (* prüfe auf gültige offset-vorgabe *)
		error_code := 255;
		step := 30000; (* Beenden *)
	ELSIF FSD.OFFSET <> file_position THEN
		command := 5; (* File-Seek *)
		seek_position := FSD.OFFSET;
		seek_mode := 0; (* Seek from beginning of file *)
		step := 210;
	ELSE
		step := 300;
	END_IF;

210: (* File Seek *)
	IF command = 0 THEN
		file_position := seek_position;
		IF error THEN
			step := 30000; (* Beenden *)
		ELSE
			step := 300;
		END_IF;
	END_IF;

300: (* Read or Write ? *)
	IF FSD.MODE = 1 THEN
		step := 400; (* Read *)
	ELSE
		step := 500; (* Write *)
	END_IF;

400: (* File Read *)
	IF UINT_TO_UDINT(PT.SIZE) > buf_size THEN (* Leselänge auf Buffergroesse begrenzen *)
		read_max_length := buf_size;
	ELSE
		read_max_length := UINT_TO_UDINT(PT.SIZE);
	END_IF;

	IF read_max_length > buf_size THEN
		read_max_length := buf_size;  (* Leselänge auf Buffergroesse begrenzen *)
	END_IF;

	(* Leselänge an Dateilänge anpassen *)
	IF file_position + read_max_length > FSD.FILE_SIZE THEN
		read_max_length := FSD.FILE_SIZE - file_position;
	END_IF;

	IF read_max_length > 0 THEN
		command := 3; (* File_Read *)
		step := 410;
	ELSE
		PT.SIZE := UINT#0;
		step := 30000; (* Beenden *)
	END_IF;

410: (* File Read *)
	IF command = 0 THEN
		PT.SIZE := UDINT_TO_UINT(length_read);
		IF NOT Error THEN
			file_position := file_position + length_read; (* aktueller File_Position korrigieren *)
			FSD.OFFSET := file_position;
		END_IF;
		step := 30000; (* Beenden *)
	END_IF;

500: (* File Write *)
	IF UINT_TO_UDINT(PT.SIZE) > buf_size THEN (* Schreiblänge auf Buffergroesse begrenzen *)
		write_length := buf_size;
	ELSE
		write_length := UINT_TO_UDINT(PT.SIZE);
	END_IF;

	IF write_length > 0 THEN
		command := 4; (* File_Write *)
		step := 510;
	ELSE
		step := 30000; (* Beenden *)
	END_IF;

510:
	IF command = 0 THEN
		IF NOT Error THEN
			file_position := file_position + length_written; (* aktueller File_Position korrigieren *)
			FSD.OFFSET := file_position;
			IF file_position > FSD.FILE_SIZE THEN (* Datei ist groesser geworden *)
				FSD.FILE_SIZE := file_position;
			END_IF;
		END_IF;
		step := 30000; (* Beenden *)
	END_IF;

 (* --------------------------------------------- *)

30000: (* Befehl fertig *)
	FSD.MODE := 0;
	FSD.ERROR := error_code;
	step := 0;

	(* ---------------- Debug-Message -----------------------*)
	(*IF _debug_enable THEN
		LOG_CL.NEW_MSG := 'FS: File_Stop: File ~1, error ~7, code ~8';
		LOG_CL.PRINTF[1]  := used_filename;
		LOG_CL.PRINTF[7]  := INT_TO_STRING(BOOL_TO_INT(error));
		LOG_CL.PRINTF[8]  := BYTE_TO_STRING(error_code);
		FB_LOG_MESSAGE();
	END_IF;*)
	(* --------------------------------------------- *)

32000:
	close_time := T#0s; (* Timer stoppen *)
	IF handle > 0 THEN
		command := 2; (* File_Close ausführen *)
	END_IF;
	step := 32100;

32100:
	IF command = 0 THEN (* File Close beendet *)
		(* Filedaten ablöschen *)
		FSD.FILE_OPEN := FALSE;
		file_position := 0;
		FSD.FILE_SIZE := 0;
		FSD.OFFSET := 0;
		used_filename := '';
		handle := 0;

		(* File_Name wurde fliegend geändert ? *)
		IF file_change THEN
			file_change := FALSE;
			step := 0;
		ELSE
			step := 30000;
		END_IF;
	END_IF;

END_CASE;

(* 1 = file_open
   2 = file_close
   3 = file_read
   4 = file_write
   5 = file_seek
   6 = file_tell
   7 = file_remove
*) 

X(bExecute := FALSE); (* Zyklischer FW_AdsRdWrt Aufruf *)

(* ------------ File Open ------------- *)
IF command = 1 THEN
	IF NOT para THEN
		para := TRUE;
		X(	nIdxGrp := 120, (* SYSTEMSERVICE_FOPEN *)
			nidxOffs := open_mode,
			cbWriteLen := SIZEOF(FSD.FILENAME),
			pWriteBuff := ADR(FSD.FILENAME),
			cbReadLen := SIZEOF(tmpDW),
			pReadBuff := ADR(tmpDW),
			bExecute := TRUE
			);
	ELSIF X.bBusy = FALSE THEN
		para := FALSE;
		error := X.bError;
		error_code := SEL(error,0,UDINT_TO_BYTE(X.nErrId + 16#10));

		IF X.cbRead >= SIZEOF(tmpDW) THEN
			open_handle := UDINT_TO_UINT(tmpDW);
		ELSE
			open_handle := 0;
		END_IF;
		command := 0;

		(* ---------------- Debug-Message -----------------------*)
		(*IF _debug_enable THEN
			LOG_CL.NEW_MSG := 'FS: Open: File ~1, handle ~2 , mode ~3 , error ~7, code ~8';
			LOG_CL.PRINTF[1] := FSD.FILENAME;
			LOG_CL.PRINTF[2] := DWORD_TO_STRING(open_handle);
			LOG_CL.PRINTF[3] := DWORD_TO_STRING(open_mode);
			LOG_CL.PRINTF[7] := INT_TO_STRING(BOOL_TO_INT(error));
			LOG_CL.PRINTF[8] := BYTE_TO_STRING(error_code);
			FB_LOG_MESSAGE();
		END_IF;*)
		(* -----------------------------------------------------------------*)
	END_IF;
END_IF;

(* ----------- File Close ------------- *)
IF command = 2 THEN
	IF NOT para THEN
		para := TRUE;
		X(	nIdxGrp := 121, (* SYSTEMSERVICE_FCLOSE *)
			nidxOffs := handle,
			cbWriteLen := 0,
			pWriteBuff := 0,
			cbReadLen := 0,
			pReadBuff := 0,
			bExecute := TRUE
			);
	ELSIF X.bBusy = FALSE THEN
		para := FALSE;
		error := X.bError;
		error_code := SEL(error,0,UDINT_TO_BYTE(X.nErrId + 16#30));
		command := 0;
		(* ---------------- Debug-Message -----------------------*)
		(*IF _debug_enable THEN
			LOG_CL.NEW_MSG := 'FS: Close: File ~1, error ~7, code ~8';
			LOG_CL.PRINTF[1] := used_filename;
			LOG_CL.PRINTF[7] := INT_TO_STRING(BOOL_TO_INT(error));
			LOG_CL.PRINTF[8] := BYTE_TO_STRING(error_code);
			FB_LOG_MESSAGE();
		END_IF;*)
		(* -----------------------------------------------------------------*)
	END_IF;
END_IF;

(* ------------ File Read ------------- *)
IF command = 3 THEN
	IF NOT para THEN
		para := TRUE;
		X(	nIdxGrp := 122, (* SYSTEMSERVICE_FREAD *)
			nidxOffs := handle,
			cbWriteLen := 0,
			pWriteBuff := 0,
			cbReadLen := read_max_length,
			pReadBuff := ADR(PT.BUFFER),
			bExecute := TRUE
			);
	ELSIF X.bBusy = FALSE THEN
		length_read := X.cbRead;
		para := FALSE;
		error := X.bError;
		error_code := SEL(error,0,UDINT_TO_BYTE(X.nErrId + 16#40));
		command := 0;

		(* ---------------- Debug-Message -----------------------*)
		(*IF _debug_enable THEN
			LOG_CL.NEW_MSG := 'FS: Read: File ~1, soll ~2,ist ~3 ,error ~7, code ~8';
			LOG_CL.PRINTF[1] := used_filename;
			LOG_CL.PRINTF[2] := UDINT_TO_STRING(read_max_length);
			LOG_CL.PRINTF[3] := UDINT_TO_STRING(length_read);
			LOG_CL.PRINTF[7] := INT_TO_STRING(BOOL_TO_INT(error));
			LOG_CL.PRINTF[8] := BYTE_TO_STRING(error_code);
			FB_LOG_MESSAGE();
		END_IF;*)
		(* -----------------------------------------------------------------*)
	END_IF;
END_IF;

(* ------------ File Write ------------- *)
IF command = 4 THEN
	IF NOT para THEN
		para := TRUE;
		X(	nIdxGrp := 123, (* SYSTEMSERVICE_FWRITE *)
			nidxOffs := handle,
			cbWriteLen := write_length,
			pWriteBuff := ADR(PT.BUFFER),
			cbReadLen := SIZEOF(length_written),
			pReadBuff := ADR(length_written),
			bExecute := TRUE
			);
	ELSIF X.bBusy = FALSE THEN
		para := FALSE;
		error := X.bError;
		error_code := SEL(error,0,UDINT_TO_BYTE(X.nErrId + 16#50));
		command := 0;

		(* ---------------- Debug-Message -----------------------*)
		(*IF _debug_enable THEN
			LOG_CL.NEW_MSG := 'FS: Write: File ~1, soll ~2,ist ~3 ,error ~7, code ~8';
			LOG_CL.PRINTF[1] := used_filename;
			LOG_CL.PRINTF[2] := UDINT_TO_STRING(write_length);
			LOG_CL.PRINTF[3] := UDINT_TO_STRING(length_written);
			LOG_CL.PRINTF[7] := INT_TO_STRING(BOOL_TO_INT(error));
			LOG_CL.PRINTF[8] := BYTE_TO_STRING(error_code);
			FB_LOG_MESSAGE();
		END_IF;*)
		(* -----------------------------------------------------------------*)
	END_IF;
END_IF;

(* ------------ File Seek ------------- *)
IF command = 5 THEN
	IF NOT para THEN
		para := TRUE;
		seek_data[0] := UDINT_TO_DINT(seek_position);
		seek_data[1] := INT_TO_DINT(seek_mode);

		X(	nIdxGrp := 124, (* SYSTEMSERVICE_FSEEK *)
			nidxOffs := handle,
			cbWriteLen := SIZEOF(seek_data),
			pWriteBuff := ADR(seek_data),
			cbReadLen := 0,
			pReadBuff := 0,
			bExecute := TRUE
			);
	ELSIF X.bBusy = FALSE THEN
		para := FALSE;
		error := X.bError;
		error_code := SEL(error,0,UDINT_TO_BYTE(X.nErrId + 16#60));
		command := 0;

		(* ---------------- Debug-Message -----------------------*)
		(*IF _debug_enable THEN
			LOG_CL.NEW_MSG := 'FS: Seek: File ~1,pos ~3 ,error ~7, code ~8';
			LOG_CL.PRINTF[1] := used_filename;
			LOG_CL.PRINTF[3] := UDINT_TO_STRING(seek_position);
			LOG_CL.PRINTF[7] := INT_TO_STRING(BOOL_TO_INT(error));
			LOG_CL.PRINTF[8] := BYTE_TO_STRING(error_code);
			FB_LOG_MESSAGE();
		END_IF;*)
		(* -----------------------------------------------------------------*)
	END_IF;
END_IF;

(* ------------ File Tell ------------- *)
IF command = 6 THEN
	IF NOT para THEN
		para := TRUE;
		X(	nIdxGrp := 125, (* SYSTEMSERVICE_FTELL *)
			nidxOffs := handle,
			cbWriteLen := 0,
			pWriteBuff := 0,
			cbReadLen := SIZEOF(tell_position),
			pReadBuff := ADR(tell_position),
			bExecute := TRUE
			);
	ELSIF X.bBusy = FALSE THEN
		para := FALSE;
		error := X.bError;
		error_code := SEL(error,0,UDINT_TO_BYTE(X.nErrId + 16#70));
		command := 0;

		(* ---------------- Debug-Message -----------------------*)
		(*IF _debug_enable THEN
			LOG_CL.NEW_MSG := 'FS: Tell: File ~1, pos ~3 ,error ~7, code ~8';
			LOG_CL.PRINTF[1] := used_filename;
			LOG_CL.PRINTF[3] := UDINT_TO_STRING(tell_position);
			LOG_CL.PRINTF[7] := INT_TO_STRING(BOOL_TO_INT(error));
			LOG_CL.PRINTF[8] := BYTE_TO_STRING(error_code);
			FB_LOG_MESSAGE();
		END_IF;*)
		(* -----------------------------------------------------------------*)
	END_IF;
END_IF;

(* ------------ File Remove ------------- *)
IF command = 7 THEN
	IF NOT para THEN
		para := TRUE;
		X(	nIdxGrp := 131, (* SYSTEMSERVICE_FDELETE *)
			nidxOffs := 16#0001_0000, (* PATH_GENERIC *)
			cbWriteLen := SIZEOF(FSD.FILENAME),
			pWriteBuff := ADR(FSD.FILENAME),
			cbReadLen := 0,
			pReadBuff := 0,
			bExecute := TRUE
			);
	ELSIF X.bBusy = FALSE THEN
		para := FALSE;
		error := X.bError;
		error_code := SEL(error,0,UDINT_TO_BYTE(X.nErrId + 16#80));
		command := 0;

		(* ---------------- Debug-Message -----------------------*)
		(*IF _debug_enable THEN
			LOG_CL.NEW_MSG := 'FS: Remove: File ~1, error ~7, code ~8';
			LOG_CL.PRINTF[1] := FSD.FILENAME;
			LOG_CL.PRINTF[7] := INT_TO_STRING(BOOL_TO_INT(error));
			LOG_CL.PRINTF[8] := BYTE_TO_STRING(error_code);
			FB_LOG_MESSAGE();
		END_IF;*)
		(* -----------------------------------------------------------------*)
	END_IF;
END_IF;

(* ---------------- Debug-Message -----------------------*)
(*IF _debug_enable THEN
	IF step_last <> step THEN
		LOG_CL.NEW_MSG := 'FS: Step: ~1';
		LOG_CL.PRINTF[1] := INT_TO_STRING(step);
		FB_LOG_MESSAGE();
	END_IF;
	step_last := step;
END_IF;*)
(* -----------------------------------------------------------------*)

(* revision history
ks	23. sep. 2010	rev 1.0
	original version
*)
END_FUNCTION_BLOCK

(* POU LOG_MSG, ST *)
FUNCTION_BLOCK LOG_MSG
(* VAR_EXTERNAL
	LOG_CL :	LOG_CONTROL;
END_VAR *)
VAR
	FB_PRINT_SF :PRINT_SF;
	idX : INT;
END_VAR

(*
version 1.0		01 mai 2010
programmer		ks
tested by		ks

LOG_MSG trägt Meldungen in den Loggingbuffer ein
*)
IF DWORD_TO_BYTE(SHL(LOG_CL.NEW_MSG_OPTION,16)) > LOG_CL.LEVEL OR NOT LOG_CL.ENABLE THEN RETURN; END_IF; (* Logging freigegeben ?*)

FB_PRINT_SF(PRINTF_DATA := LOG_CL.PRINTF,STR := LOG_CL.NEW_MSG);

IF LOG_CL.RESET THEN (* Logeinträge löschen *)
	LOG_CL.RESET := FALSE;
	LOG_CL.RING_MODE := FALSE;
	LOG_CL.IDX := 0;
	LOG_CL.UPDATE_COUNT := LOG_CL.UPDATE_COUNT + UINT#1; (* UpdateCount erhöhen *)
END_IF;

IF LOG_CL.SIZE > 0 THEN (* size wert ist eingetragen *)
	IF LEN(LOG_CL.NEW_MSG) > 0 THEN (* Meldung in Puffer eintragen *)
		IF (LOG_CL.IDX >= LOG_CL.SIZE) THEN
			LOG_CL.RING_MODE := TRUE; (* bei Überlauf = Ringbuffermodus *)
			LOG_CL.IDX := 0; (* wieder auf arrayanfang positionieren *)
		END_IF;

		LOG_CL.UPDATE_COUNT := LOG_CL.UPDATE_COUNT + UINT#1; (* UpdateCount erhöhen *)
		LOG_CL.IDX := LOG_CL.IDX + INT#1; (* nächste freie Position *)
		idx := LOG_CL.IDX; (* lade aktuelle Log-Puffer Positition *)
		LOG_CL.MSG[idx] := LOG_CL.NEW_MSG; (* neuen Log-String in puffer ablegen  *)
		LOG_CL.MSG_OPTION[idx] := LOG_CL.NEW_MSG_OPTION; (* neue Log-String Option in puffer ablegen  *)
		LOG_CL.NEW_MSG := ''; (* letzten Log-String löschen *)
	END_IF;
END_IF;
END_FUNCTION_BLOCK

(* POU PRINT_SF, ST *)
FUNCTION_BLOCK PRINT_SF
VAR_IN_OUT
	PRINTF_DATA : PRINTF_DATA;
	STR : STRING(LOG_SIZE);
END_VAR
VAR
	pos : INT;
	c : INT;
	src : STRING(1) := '~';
	run : BOOL;
END_VAR

(*

version 1.0 		14. aug. 2009
programmer 	ks
tested by		ks

PRINTF erzeugt aus einem Parameterstring und den übergebenen Parameterdaten einen Text
*)
IF LEN(STR) > 0 THEN
	run := TRUE;

	WHILE (run) DO
		pos := FIND(STR,src);
		PRINTF_DATA[10] := '';

		IF pos = 0 THEN
			run:= FALSE;
		ELSE
			c := CODE(STR:=STR,POS:=pos + 1);
			IF ISC_NUM(INT_TO_BYTE(c)) THEN
				c := c - 48; (* notwendig weil innerhalb einer indexangabe nur eine var stehen darf *)
				PRINTF_DATA[10] := PRINTF_DATA[c]; (* Kommando 1-9 ergibt Parameterindex 1-9 *)
				(* Parameter gegen Text tauschen *)
			END_IF;
			IF LEN(PRINTF_DATA[10]) + LEN(STR) > LOG_SIZE THEN
				PRINTF_DATA[10] := '..';
			END_IF;
			(* pcworx: aus und eingangsstring muss verschieden sein *)
			PRINTF_DATA[11] := STR;
			STR := REPLACE(PRINTF_DATA[11],PRINTF_DATA[10],2,pos);
		END_IF;
	END_WHILE;
END_IF;

(* revision history

ks	14. aug. 2009	rev 1.0
	original version

*)
END_FUNCTION_BLOCK

(* POU CSV_PARSER_FILE_DEMO, ST *)
PROGRAM CSV_PARSER_FILE_DEMO
VAR CONSTANT
	 line_cnt : INT:=2;
	 col_cnt : INT:=4;
END_VAR
VAR
	CPF : CSV_PARSER_FILE;
	FS : FILE_SERVER;
	FSD : FILE_SERVER_DATA;
	PT : NETWORK_BUFFER;
	filename : STRING;
	value :	STRING(STRING_LENGTH);
	sep : BYTE;
	step : INT;
	result : BYTE;
	offset : UDINT;
	run : BYTE;
	done : BOOL;
	value_real : REAL;
	cnt : INT;
	line : INT;
	idx : INT;
	data : ARRAY [1..line_cnt, 1..col_cnt] OF REAL;
	FB_LOG_MESSAGE : LOG_MSG;
END_VAR
(* Demo-Programm: CSV-Datei mittels Enumeration auswerten

die groesse des arrays kann mittels konstanten line_cnt und col_cnt angepasst werden

 ----- den nachfolgenden Textblock als datei "csv.txt" auf der sps ablegen ---
10.45,20,30,40.8
115,3450.2123,456,123.1
---------------------------------------------------------------------------------*)

CASE step OF

00:	IF NOT done THEN
		filename := 'd:\pxc\oscat\network\csv.txt'; (* File_Daten einrichten *)
		OFFSET := 0; (* Start Offset vorgeben *)
		FSD.AUTO_CLOSE := T#0ms; (* kein Automatisches schliessen *)
		sep :=44; (* Trennzeichen , *)
		run := 1; (* Element suchen *)
		cnt := 0;
		step := 20;
	END_IF;

20:	IF run = 0 THEN (* kein Befehl mehr aktiv ? *)
		(* ---------------------- Debug-Message ----------------------------*)
		IF LOG_CL.ENABLE THEN
			LOG_CL.NEW_MSG := 'CPFD: /value >~2< /offset ~3 /Run ~4 /Result ~5';
			LOG_CL.PRINTF[2] := value;
			LOG_CL.PRINTF[3] := UDINT_TO_STRING(OFFSET);
			LOG_CL.PRINTF[4] := BYTE_TO_STRING(run);
			LOG_CL.PRINTF[5] := BYTE_TO_STRING(result);
			FB_LOG_MESSAGE();
		END_IF;
		(* -----------------------------------------------------------------*)

		run := 1; (*  nächstes Element suchen  *)

		IF result = 1 OR result = 2 THEN
			(* automatische konvertierung in real ausführen *)
			IF LEN(value) <= 20 THEN
				value_real := FLOAT_TO_REAL(FLT:=value);
			ELSE
				value_real := 0.0;
			END_IF;

			cnt := cnt + 1;
			IF cnt <= line_cnt * col_cnt THEN
				line := (cnt / col_cnt) + 1;
				idx := (cnt MOD col_cnt);
				data[line,idx] := value_real; (* Daten in Array eintragen *)
			END_IF;

		ELSIF result = 10 THEN (* nichts mehr gefunden *)
			run := 0; (* keine weitere INI Auswertung erwünscht *)
			FSD.MODE := 5; (* Datei schliessen *)
			step := 30;
		END_IF;
	END_IF;

30:	IF FSD.MODE = 0 THEN (* Befehl Datei schliessen beendet *)
		step := 0;
		done := TRUE;
	END_IF;

END_CASE;

CPF(SEP:=sep,FILENAME:=FILENAME,FSD:=FSD,RUN:=run,OFFSET:=OFFSET,VALUE:=value,PT:=PT,RESULT=>result); (* CSV PARAMETER FILE *)
FS(FSD:=FSD,PT:=PT); (* FILE_SERVER *)
END_PROGRAM

(* POU CSV_PARSER_FILE, ST *)
FUNCTION_BLOCK CSV_PARSER_FILE
VAR_INPUT
	SEP : BYTE;
END_VAR
VAR_IN_OUT
	FILENAME : STRING;
	FSD : FILE_SERVER_DATA;
	RUN : BYTE;
	OFFSET : UDINT;
	VALUE : STRING(STRING_LENGTH);
	PT	: NETWORK_BUFFER;
END_VAR
VAR_OUTPUT
	RESULT : BYTE;
END_VAR
VAR
	i : UDINT;
	state : BYTE;
	e : BYTE;
	mode : BYTE;
	step : INT;
	c : BYTE;
	v_add : BYTE;
	eof : BOOL;
	pv : POINTER TO BYTE;
	pve : DWORD;
	watchdog : TON;
	x : BOOL;
	FB : FILE_BLOCK;

	(*FB_LOG_MESSAGE : LOG_MSG;
	_debug_enable : BOOL := FALSE;
	step_last : INT;*)
END_VAR

(*
version 1.0		01. oct. 2010
programmer 		ks
tested by			ks

CSV_PARSER_FILE liefert die Elemente oder Zeilen einer Textdatei.

--------------------------------------

RUN Mode
00 = kein Befehl aktiv
01 = Element suchen

Result Codes
01 = Element gefunden
02 = Element und Zeilenende erkannt
05 = Befehl in Arbeit (Busy)
10 = nichts gefunden - Daten-Ende erreicht

State Codes
01 = Element gefunden
02 = Element und Zeilenende erkannt
05 = Befehl in Arbeit (Busy)
10 = nichts gefunden - Daten-Ende erreicht

*)
IF RUN > 0 THEN

	IF state = 0 THEN (* Auswertung neu beginnen *)
		pv := ADR(VALUE);
		pv^ := 0; (* VALUE = '' *)
		pve := pv + INT_TO_DWORD(STRING_LENGTH);
		i := OFFSET;
		RESULT := 0;
		state := 5; (* Befehl in Arbeit (Busy) *)
		step := 0; (* Auswertung neu beginnen *)

		(* ---------------- Debug-Message -----------------------*)
		(*IF _debug_enable THEN
			LOG_CL.NEW_MSG := 'CPF: Startindex: ~1';
			LOG_CL.PRINTF[1] := UDINT_TO_STRING(i);
			FB_LOG_MESSAGE();
		END_IF;*)
		(* -----------------------------------------------------------------*)

	END_IF;

	watchdog(IN:=FALSE,PT:=T#1ms); (* Timer neustarten *)
	watchdog.IN := TRUE;

	WHILE (state = 5) DO (* Schleife solange kein Ergebnis *)

		mode := 1;
		FB(MODE:=mode,FSD:=fsd,PT:=PT,FILENAME:=FILENAME,POS:=i );
		e:=FB.ERROR;
		c:=FB.DATA;

		eof := i + 1 = FSD.FILE_SIZE; (* End of File *)

		(* ---------------- Debug-Message -----------------------*)
		(*IF _debug_enable THEN
			LOG_CL.NEW_MSG := 'CPF: mode: ~1, error: ~2 , >~7<>~3< ~4 step ~5 index ~6';
			LOG_CL.PRINTF[1] := BYTE_TO_STRING(mode);
			LOG_CL.PRINTF[2] := BYTE_TO_STRING(e);
			LOG_CL.PRINTF[3] := BYTE_TO_STRING(c);
			LOG_CL.PRINTF[4] := BOOL_TO_STRING(eof);
			LOG_CL.PRINTF[5] := INT_TO_STRING(step);
			LOG_CL.PRINTF[6] := UDINT_TO_STRING(i);
			LOG_CL.PRINTF[7] := CHR_TO_STRING(c);
			FB_LOG_MESSAGE();
		END_IF;*)
		(* -----------------------------------------------------------------*)
		watchdog(); (* Timer aktualisieren *)

		IF mode > 0 OR watchdog.Q THEN (* Baustein noch aktiv, oder watchdog ausgelöst *)
			state := 5;
			EXIT;
		ELSIF e > 0 THEN (* File_error oder kein weiteres zeichen vorhanden *)
			state := 10; (* nichts gefunden - Daten-Ende erreicht *)
			EXIT;
		ELSE

			v_add := 0;

			IF c = SEP THEN (* Neues Element erkannt *)
				state := 1;
				x := TRUE;
			ELSIF c >= 32 THEN (* Element erkannt *)
				v_add := c; (* Zeichen ablegen *)
				IF eof THEN
					state := 2; (* Element und Zeilenende erkannt *)
				ELSE
					x := TRUE;
				END_IF;
			ELSE
				IF x THEN
					state := 2; (* Element und Zeilenende erkannt *)
					x := FALSE;
				END_IF;
			END_IF;

			IF v_add > 0  AND pv < pve THEN (* Zeichen zu Value-String hinzufügen *)
				pv^ := v_add; (* Zeichen eintragen *)
				pv := pv + 1;
				pv^ := 0; (* String-Terminierung eintragen *)
			END_IF;

			i := i + 1; (* Datenzeiger erhöhen *)

		END_IF;
	END_WHILE;

	CASE state OF
	01:	(* Element gefunden *)
		RESULT := 1; (* Element gefunden *)
		OFFSET := i; (* Offset uebernehmen *)
		RUN := 0;
		state := 0;
	02:	(* Element gefunden *)
		RESULT := 2; (* Element und Zeilenende erkannt *)
		OFFSET := i; (* Offset uebernehmen *)
		RUN := 0;
		state := 0;

	05:	RESULT := 5; (* in Arbeit *)

	10:	(* Indexüberschreitung - Bufferende *)
		RESULT := 10; (* nichts gefunden - Datenende erreicht *)
		OFFSET := i; (* Offset uebernehmen *)
		RUN := 0;
		state := 0;
	END_CASE;

	(* ---------------- Debug-Message -----------------------*)
	(*IF _debug_enable THEN
		LOG_CL.NEW_MSG := 'CPF: intern Result ~1 , state ~2, step ~3 , offset ~4, run ~5';
		LOG_CL.PRINTF[1] := BYTE_TO_STRING(RESULT);
		LOG_CL.PRINTF[2] := BYTE_TO_STRING(state);
		LOG_CL.PRINTF[3] := INT_TO_STRING(step);
		LOG_CL.PRINTF[4] := UDINT_TO_STRING(OFFSET);
		LOG_CL.PRINTF[5] := BYTE_TO_STRING(RUN);
		FB_LOG_MESSAGE();
	END_IF;*)
	(* -----------------------------------------------------------------*)

END_IF;

(* ---------------- Debug-Message -----------------------*)
(*IF _debug_enable THEN
	IF step_last <> step THEN
		LOG_CL.NEW_MSG := 'CPF: Step: ~1';
		LOG_CL.PRINTF[1]  := INT_TO_STRING(step);
		FB_LOG_MESSAGE();
	END_IF;
	step_last := step;
END_IF;*)
(* -----------------------------------------------------------------*)

(* revision history
ks	01. oct. 2010	rev 1.0
	original version
*)
END_FUNCTION_BLOCK

(* POU FILE_BLOCK, ST *)
FUNCTION_BLOCK FILE_BLOCK
VAR_IN_OUT
	MODE : BYTE;
	FILENAME : STRING;
	FSD : FILE_SERVER_DATA;
	PT : NETWORK_BUFFER;
END_VAR
VAR_INPUT
	POS : UDINT;
END_VAR
VAR_OUTPUT
	ERROR : BYTE;
	DATA : BYTE;
END_VAR
VAR
	step : INT;
	i : INT;
	data_start : UDINT;
	data_stop : UDINT;

	(*FB_LOG_MESSAGE : LOG_MSG;
	_debug_enable : BOOL := TRUE;*)
END_VAR

(*
version 1.0		23. sep. 2010
programmer 		ks
tested by			ks

FILE_BLOCK liefert das angeforderte BYTE einer Datei durch einlesen von möglichst grossen Datenblöcken
*)
CASE step OF
0:	IF MODE > 0 THEN
		ERROR := 0;
		IF FSD.FILE_OPEN AND (FSD.FILE_SIZE = 0 OR POS >= FSD.FILE_SIZE) THEN
			ERROR := 255;
			MODE := 0;
		ELSIF POS < data_start OR POS > data_stop OR NOT FSD.FILE_OPEN THEN (* Daten lesen notwendig *)
			FSD.FILENAME := FILENAME;
			FSD.MODE := 1; (* open + read *)
			FSD.OFFSET := POS;
			PT.SIZE := 65535; (* maximale anzahl lesen *);
			data_start := 0;
			data_stop := 0;
			step := 10;
		ELSE (* Daten sind im Buffer vorhanden *)
			i := UDINT_TO_INT(POS - data_start); (* index berechnen *)
			DATA := PT.BUFFER[i];
			MODE := 0;
			(* ---------------------- Debug-Message ----------------------------*)
			(*IF _debug_enable THEN
				LOG_CL.NEW_MSG := 'FB: Pos: ~1 Byte: ~2 >~3<';
				LOG_CL.PRINTF[1] := UDINT_TO_STRING(POS);
				LOG_CL.PRINTF[2] := BYTE_TO_STRING(DATA);
				LOG_CL.PRINTF[3] := CHR_TO_STRING(DATA);
				FB_LOG_MESSAGE();
			END_IF;*)
			(* -----------------------------------------------------------------*)
		END_IF;
	END_IF;

10:	IF FSD.MODE = 0 THEN (* Befehl beendet *)
		IF FSD.ERROR > 0 THEN
			ERROR := FSD.ERROR; (* Fehler ausgeben *)
			MODE := 0;
		ELSE
			data_start := POS;
			data_stop := POS + UINT_TO_UDINT(PT.SIZE) - 1;
		END_IF;
		step := 0;
	END_IF;
END_CASE;

(* revision history
ks	23. sep. 2010	rev 1.0
	original version
*)
END_FUNCTION_BLOCK

(* POU DLOG_FILE_CSV_FTP_DEMO, CFC *)
PROGRAM DLOG_FILE_CSV_FTP_DEMO
VAR
	RTC_2: RTC_2;
	x : DLOG_DATA;
	DLOG_STORE_FILE_CSV : DLOG_STORE_FILE_CSV;
	CLK_PRG: CLK_PRG;
	cur_dt: DT;
	enable: BOOL;
	rtc_set : BOOL := TRUE;

	trig_t : UDINT := 6;
	trig_m : BOOL;

	x1: DLOG_DT;
	x2 : DLOG_REAL;
	x3 : DLOG_DINT;
	GEN_SIN_1: GEN_SIN;
	COUNT_DR: COUNT_DR;

	DLOG_FILE_TO_FTP: DLOG_FILE_TO_FTP;
	ftp_done: BOOL;
	ftp_busy: BOOL;
	ftp_error_c: DWORD;
	ftp_error_t: BYTE;
	ftp_url: STRING := 'ftp://581920:123456@oscat.atwebpages.com:2000/subordner/';
	ftp_activ: BOOL := FALSE;
	ftp_delete: BOOL := TRUE;
	ftp_retry: INT := 0;
	ftp_retry_time: TIME := T#60s;
	ftp_timeout: TIME := T#30s;

END_VAR
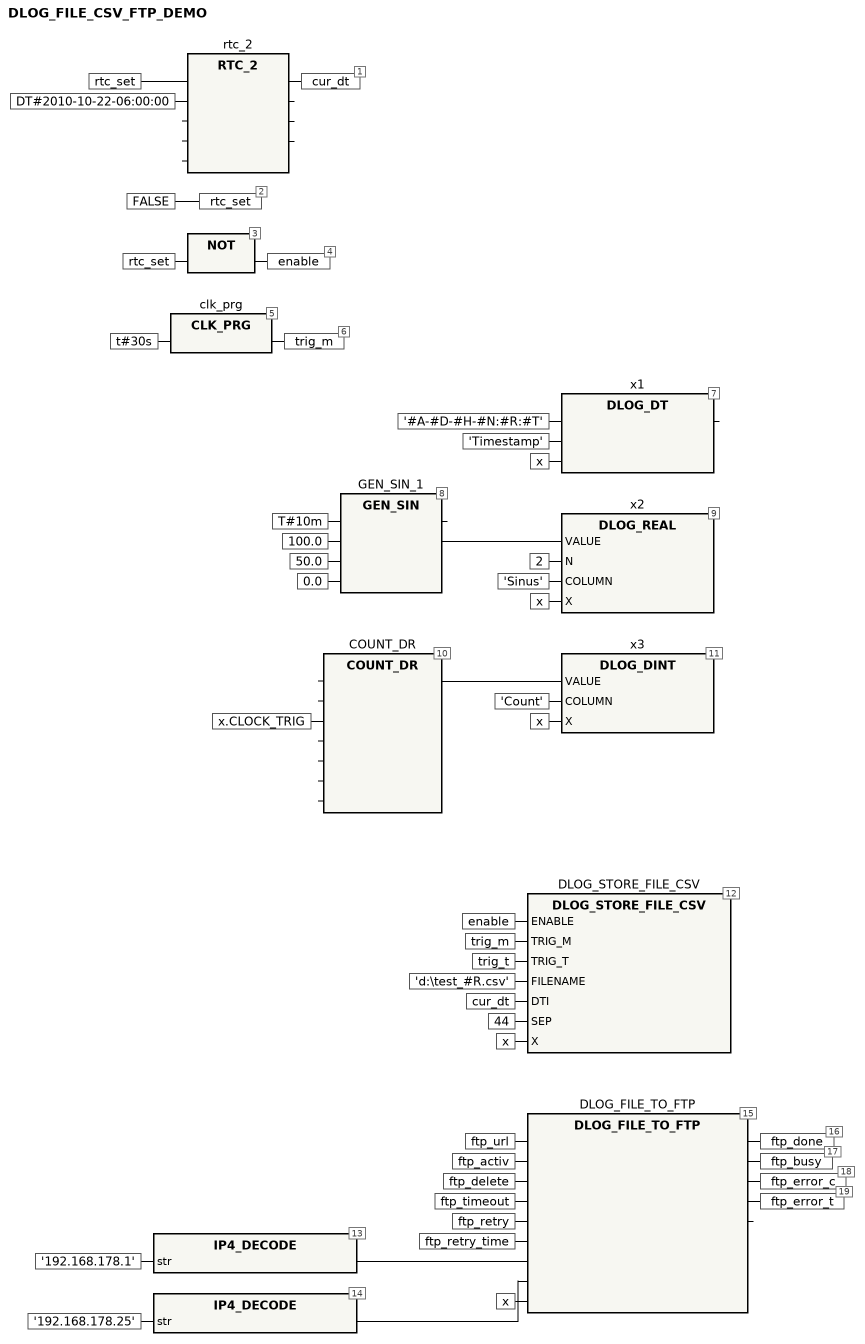
_CFC_ (* Continuous Function Chart, elements in execution order *)
#0 rtc_2:RTC_2(rtc_set, DT#2010-10-22-06:00:00, -, -, -)
#1 cur_dt <= #0.out 1
#2 rtc_set <= FALSE
#3 NOT(rtc_set)
#4 enable <= #3
#5 clk_prg:CLK_PRG(t#30s)
#6 trig_m <= #5
#7 x1:DLOG_DT('#A-#D-#H-#N:#R:#T', 'Timestamp', x)
#8 GEN_SIN_1:GEN_SIN(T#10m, 100.0, 50.0, 0.0)
#9 x2:DLOG_REAL(VALUE: #8.out 2, N: 2, COLUMN: 'Sinus', X: x)
#10 COUNT_DR:COUNT_DR(-, -, x.CLOCK_TRIG, -, -, -, -)
#11 x3:DLOG_DINT(VALUE: #10, COLUMN: 'Count', X: x)
#12 DLOG_STORE_FILE_CSV:DLOG_STORE_FILE_CSV(ENABLE: enable, TRIG_M: trig_m, TRIG_T: trig_t, FILENAME: 'd:\test_#R.csv', DTI: cur_dt, SEP: 44, X: x)
#13 IP4_DECODE(str: '192.168.178.1')
#14 IP4_DECODE(str: '192.168.178.25')
#15 DLOG_FILE_TO_FTP:DLOG_FILE_TO_FTP(ftp_url, ftp_activ, ftp_delete, ftp_timeout, ftp_retry, ftp_retry_time, #13, #14, x)
#16 ftp_done <= #15.out 1
#17 ftp_busy <= #15.out 2
#18 ftp_error_c <= #15.out 3
#19 ftp_error_t <= #15.out 4
_END_CFC_
END_PROGRAM

(* POU DLOG_STORE_FILE_CSV, ST *)
FUNCTION_BLOCK DLOG_STORE_FILE_CSV
VAR_IN_OUT
	X : DLOG_DATA;
END_VAR
VAR_INPUT
	ENABLE : BOOL;
	TRIG_M : BOOL;
	TRIG_T : UDINT;
	FILENAME : STRING;
	DTI : DT;
	SEP : BYTE;
END_VAR
VAR_OUTPUT
END_VAR
VAR
	FS : FILE_SERVER;
	FSD : FILE_SERVER_DATA;
	PT : NETWORK_BUFFER;
	UCB : UNI_CIRCULAR_BUFFER;
	ra : BOOL;
	trig_m_last : BOOL;
	dti_last : DT := DT#2070-02-06-06:28:15;
	enable_last : BOOL;
	fn_last : STRING;
	fn : STRING;
	init : BOOL;
	step: INT;
	idx : INT;
	log_stop : BOOL;
END_VAR

(*
version 1.0		01. jan. 2011
programmer		ks
tested by			ks

DLOG_STORE_FILE_CSV der Baustein schreibt die DLOG Parameter in einen lokale Datei im CSV-Format
*)
X.DTI := DTI; (* Datum / Zeit eintragen *)
IF DTI <> dti_last THEN
	X.CLOCK_TRIG := TRUE;
	dti_last := DTI;
ELSE
	X.CLOCK_TRIG := FALSE;
END_IF;

IF X.ADD_HEADER = FALSE THEN (* wenn add-header und add-data gleichzeitig ansteht, dann add-data einen zyklus länger anstehen lassen *)
	X.ADD_DATA := FALSE;
END_IF;
X.ADD_HEADER := FALSE;

IF ENABLE THEN
	IF X.CLOCK_TRIG THEN
		fn := DT_TO_STRF(DTI, 0, FILENAME, 0); (* automatische Dateinamen generierung *)
		IF TRIG_T > 0 THEN (* automatischer Trigger *)
			ra := DT_TO_UDINT(DTI) MOD TRIG_T = 0;
		END_IF;
	ELSE
		ra := FALSE;
	END_IF;
	IF (TRIG_M AND NOT trig_m_last) OR ra THEN (* manueller oder automatischer Trigger *)
		X.ADD_DATA := TRUE; (* Daten loggen *)
	END_IF;
	IF NOT init THEN
		init := TRUE;
		X.ADD_HEADER := TRUE; (* Spaltenüberschriften übernehmen *)
	END_IF;
END_IF;

IF (NOT ENABLE AND enable_last) OR (fn <> fn_last AND step > 0) THEN (* Neg. Flanke ENABLE - Log Stop *)
	fn_last := fn;
	X.UCB.D_HEAD := WORD#16#FF00;
	X.UCB.D_MODE := 1;
	UCB(DATA:=X.UCB); (* Element schreiben *)
	X.ADD_HEADER := TRUE; (* Spaltenüberschriften übernehmen *)
END_IF;

CASE step OF

00:	IF ENABLE THEN
		fn_last := fn;
		FSD.FILENAME := fn; (* Dateiname *)
		FSD.OFFSET := 0; (* Start bei Dateianfang *)
		FSD.AUTO_CLOSE := T#0s; (* Auto-Close *)
		step := 20;
	END_IF;

20:	IF X.UCB.BUF_COUNT > 0 THEN (* Einträge vorhanden *)
		X.UCB.D_MODE := 10;
		UCB(DATA:=X.UCB); (* Element lesen , aber noch nicht entfernen *)
		IF X.UCB.D_HEAD = WORD#16#FF00 THEN (* LOG_STOP Command *)
			X.UCB.D_MODE := 11;
			UCB(DATA:=X.UCB); (* Element entfernen *)
			log_stop := TRUE;
			step := 40; (* Daten schreiben *)
		ELSIF idx + LEN(X.UCB.D_STRING) + 2 < SIZEOF(PT) THEN (* Platz für Element vorhanden ? *)
			X.UCB.D_MODE := 11;
			UCB(DATA:=X.UCB); (* Element entfernen *)
			_STRING_TO_BUFFER(STR:=X.UCB.D_STRING, POS:=idx, PT:=ADR(PT.BUFFER), SIZE:=SIZEOF(PT.BUFFER));
			idx := idx + LEN(X.UCB.D_STRING);
			IF X.ID_MAX = SHR(X.UCB.D_HEAD,8) THEN (* letztes Element einer Zeile *)
				PT.BUFFER[idx] := 16#0D;
				idx := idx + 1;
				PT.BUFFER[idx] := 16#0A;
			ELSE
				PT.BUFFER[idx] := SEP;
			END_IF;
			idx := idx + 1;
		ELSE
			step := 40; (* Daten schreiben *)
		END_IF;
	END_IF;

40:	IF idx > 0 THEN (* Daten schreiben *)
		FSD.MODE := 3; (* create + write *)
		PT.SIZE := idx; (* Datenlänge eintragen *)
		idx := 0;
	END_IF;
	step := 60;

60:	IF FSD.MODE = 0 THEN
		IF log_stop THEN
			log_stop := FALSE;
			FSD.MODE := 5; (* Datei schliessen *)
			X.NEW_FILE := FSD.FILENAME;
			X.NEW_FILE_RTRIG := FALSE;
			step := 80;
		ELSE
			step := 20;
		END_IF;
	END_IF;

80:	IF FSD.MODE = 0 THEN (* Datei schliessen beendet *)
		X.NEW_FILE_RTRIG := TRUE;
		step := 0;
	END_IF;

END_CASE;

trig_m_last := TRIG_M;
enable_last := ENABLE;
FS(FSD:=FSD,PT:=PT); (* FILE_SERVER *)

(* revision history
ks	01. jan. 2011	rev 1.0
	original version
*)
END_FUNCTION_BLOCK

(* POU UNI_CIRCULAR_BUFFER, ST *)
FUNCTION_BLOCK UNI_CIRCULAR_BUFFER
VAR_IN_OUT
	DATA : UNI_CIRCULAR_BUFFER_DATA;
END_VAR
VAR_TEMP
	tmp_dw : DWORD;
	pTmp : POINTER TO BYTE;
	n : INT;
	n1 : INT;
	n2 : INT;
	x: BYTE;
	buf_totalsize : UINT;
END_VAR
VAR CONSTANT
	HeaderSize : INT := 4;
END_VAR
VAR
	cnt : UINT;
	mode_last : INT;

	(*FB_LOG_MESSAGE : LOG_MSG;
	_debug_enable : BOOL := FALSE;*)
END_VAR

(*
version 1.0		01. jan. 2011
programmer		ks
tested by			ks

UNI_CIRCULAR_BUFFER ist ein FIFO-RING-Buffer der verschiedene Datenelemente als Byte-Array aufnehmen kann.
*)
CASE DATA.D_MODE OF

01:	x := WORD_TO_BYTE(DATA.D_HEAD); (* nur rechtes byte auswerten *)
	CASE x OF
	01:	cnt := LEN(DATA.D_STRING); (* String verarbeiten *)
		pTmp := ADR(DATA.D_STRING);
	02:	cnt := 4; (* Real verarbeiten *)
		pTmp := ADR(DATA.D_REAL);
	03:	cnt := 4; (* DWORD verarbeiten *)
		pTmp := ADR(DATA.D_DWORD);
	ELSE
		cnt := 0;
	END_CASE;

	(* ------ Daten in buffer eintragen ------ *)
	buf_totalsize := SIZEOF(DATA.BUF);

	IF (cnt + HeaderSize) > (buf_totalsize - DATA.BUF_SIZE) THEN (* genug Speicher frei ? *)
		RETURN;
	END_IF;

	mode_last := DATA.D_MODE;
	tmp_dw := SHL(WORD_TO_DWORD(DATA.D_HEAD),16) OR UINT_TO_DWORD(cnt);

	(* Header in Buffer eintragen *)
	n1 := 0;
	REPEAT
		n2 := MIN(HeaderSize - n1, buf_totalsize - DATA._Last);
		FOR n := 1 TO n2 DO
			tmp_dw := ROL(tmp_dw,8);
			data.BUF[DATA._Last] := DWORD_TO_BYTE(tmp_dw);
			DATA._Last := DATA._Last + 1;
		END_FOR;
		IF DATA._Last >= buf_totalsize THEN
			DATA._Last := 0;
		END_IF
		n1 := n1 + n2;
	UNTIL n1 >= HeaderSize
	END_REPEAT;

	(* Daten in Buffer eintragen *)
	n1 := 0;
	REPEAT
		n2 := MIN(cnt - n1, buf_totalsize - DATA._Last);
		FOR n := 1 TO n2 DO
			data.BUF[DATA._Last] := pTmp^;
			pTmp := pTmp + 1;
			DATA._Last := DATA._Last + 1;
		END_FOR;
		IF DATA._Last >= buf_totalsize THEN
			DATA._Last := 0;
		END_IF
		n1 := n1 + n2;
	UNTIL n1 >= cnt
	END_REPEAT;

	DATA.BUF_SIZE := DATA.BUF_SIZE + cnt + HeaderSize;
	DATA.BUF_COUNT := DATA.BUF_COUNT + 1;
	DATA.BUF_USED := UINT_TO_USINT(100 * DATA.BUF_SIZE / buf_totalsize); (* benützer Speicher in % *)
	DATA.D_MODE := 0;

	(*####################  DEBUG-MESSAGE  ###################################*)
	(*IF _debug_enable THEN
		LOG_CL.NEW_MSG := 'RP: ADD /HEAD ~1 / SIZE ~2 / CNT ~3 / >~4<';
		LOG_CL.PRINTF[1] := DWORD_TO_STRH(DATA.D_HEAD);
		LOG_CL.PRINTF[2] := UINT_TO_STRING(cnt);
		LOG_CL.PRINTF[3] := UINT_TO_STRING(DATA.BUF_COUNT);
		CASE x OF
		01:	LOG_CL.PRINTF[4] := DATA.D_STRING;
		02:	LOG_CL.PRINTF[4] := REAL_TO_STRING(DATA.D_REAL);
		03:	LOG_CL.PRINTF[4] := DWORD_TO_STRH(DATA.D_DWORD);
		ELSE
			LOG_CL.PRINTF[4] := '';
		END_CASE;
		FB_LOG_MESSAGE();
	END_IF;*)
	(*########################################################################*)

10:	(* ------ Daten aus buffer auslesen ------ *)
	IF DATA.BUF_COUNT = 0 THEN RETURN; END_IF;
	buf_totalsize := SIZEOF(DATA.BUF);
	DATA._GetEnd := DATA._First;(* index des ältesten eintrags merken *)
	mode_last := DATA.D_MODE;

	(* Header aus Buffer lesen *)
	n1 := 0;
	tmp_dw := 0;
	REPEAT
		n2 := MIN(HeaderSize - n1, buf_totalsize - DATA._GetEnd);
		FOR n := 1 TO n2 DO
			tmp_dw := ROL(tmp_dw,8) OR BYTE_TO_DWORD(data.BUF[DATA._GetEnd]);
			DATA._GetEnd := DATA._GetEnd + 1;
		END_FOR;
		IF DATA._GetEnd >= buf_totalsize THEN
			DATA._GetEnd := 0;
		END_IF
		n1 := n1 + n2;
	UNTIL n1 >= HeaderSize
	END_REPEAT;

	DATA._GetStart := DATA._GetEnd;
	cnt := DWORD_TO_UINT(tmp_dw AND 16#0000_FFFF);
	DATA.D_HEAD := DWORD_TO_WORD(SHR(tmp_dw,16));

	x := WORD_TO_BYTE(DATA.D_HEAD); (* nur rechtes byte auswerten *)
	CASE x OF
	01:	pTmp := ADR(DATA.D_STRING); (* String verarbeiten *)
	02:	pTmp := ADR(DATA.D_REAL); (* Real verarbeiten *)
	03:	pTmp := ADR(DATA.D_DWORD); (* DWORD verarbeiten *)
	END_CASE;

	(* Daten aus Buffer lesen *)
	n1 := 0;
	REPEAT
		n2 := MIN(cnt - n1, buf_totalsize - DATA._GetEnd);
		FOR n := 1 TO n2 DO
			pTmp^ := data.BUF[DATA._GetEnd];
			pTmp := pTmp + 1;
			DATA._GetEnd := DATA._GetEnd + 1;
		END_FOR;
		IF DATA._GetEnd >= buf_totalsize THEN
			DATA._GetEnd := 0;
		END_IF
		n1 := n1 + n2;
	UNTIL n1 >= cnt
	END_REPEAT;
	IF x = 1 THEN
		pTmp^ := 0; (* String terminieren *)
	END_IF;
	DATA.D_MODE := 0;

	(*####################  DEBUG-MESSAGE  ###################################*)
	(*IF _debug_enable THEN
		LOG_CL.NEW_MSG := 'RP: READ /HEAD ~1 / SIZE ~2 / CNT ~3 / >~4<';
		LOG_CL.PRINTF[1] := DWORD_TO_STRH(DATA.D_HEAD);
		LOG_CL.PRINTF[2] := UINT_TO_STRING(cnt);
		LOG_CL.PRINTF[3] := UINT_TO_STRING(DATA.BUF_COUNT);
		CASE x OF
		01:	LOG_CL.PRINTF[4] := DATA.D_STRING;
		02:	LOG_CL.PRINTF[4] := REAL_TO_STRING(DATA.D_REAL);
		03:	LOG_CL.PRINTF[4] := DWORD_TO_STRH(DATA.D_DWORD);
		ELSE
			LOG_CL.PRINTF[4] := '';
		END_CASE;
		FB_LOG_MESSAGE();
	END_IF;*)
	(*########################################################################*)

11:	IF mode_last = 10 THEN (* löschen nur direkt nach lesen möglich *)
		mode_last := DATA.D_MODE;
		DATA.BUF_SIZE := DATA.BUF_SIZE - cnt - HeaderSize;
		DATA.BUF_COUNT := DATA.BUF_COUNT - 1;
		DATA._First := DATA._GetEnd;
		DATA.BUF_USED := UINT_TO_USINT(100 * DATA.BUF_SIZE / SIZEOF(DATA.BUF)); (* benützer Speicher in % *)
		DATA.D_MODE := 0;

		(*####################  DEBUG-MESSAGE  ###################################*)
		(*IF _debug_enable THEN
			LOG_CL.NEW_MSG := 'RP: DEL /HEAD ~1 / SIZE ~2 / CNT ~3 / >~4<';
			LOG_CL.PRINTF[1] := DWORD_TO_STRH(DATA.D_HEAD);
			LOG_CL.PRINTF[2] := UINT_TO_STRING(cnt);
			LOG_CL.PRINTF[3] := UINT_TO_STRING(DATA.BUF_COUNT);
			CASE x OF
			01:	LOG_CL.PRINTF[4] := DATA.D_STRING;
			02:	LOG_CL.PRINTF[4] := REAL_TO_STRING(DATA.D_REAL);
			03:	LOG_CL.PRINTF[4] := DWORD_TO_STRH(DATA.D_DWORD);
			ELSE
				LOG_CL.PRINTF[4] := '';
			END_CASE;
			FB_LOG_MESSAGE();
		END_IF;*)
		(*########################################################################*)
	END_IF;

99:	(* Buffer reset - alles löschen *)
	DATA._First := 0;
	DATA._Last := 0;
	DATA._GetStart := 0;
	DATA._GetEnd := 0;
	DATA.BUF_COUNT := 0;
	DATA.BUF_SIZE := 0;
	DATA.BUF_USED := 0;
	DATA.D_STRING := '';
	DATA.D_DWORD := 0;
	DATA.D_REAL := 0.0;
	DATA.D_HEAD := 0;
	DATA.D_MODE := 0;
	mode_last := 0;
END_CASE;

(* revision history
ks	01. jan. 2011	rev 1.0
	original version
*)
END_FUNCTION_BLOCK

(* POU DLOG_DT, ST *)
FUNCTION_BLOCK DLOG_DT
VAR_IN_OUT
	X : DLOG_DATA;
END_VAR
VAR_INPUT
	FMT : STRING;
	COLUMN : STRING;
END_VAR

VAR_OUTPUT
END_VAR
VAR
	UCB : UNI_CIRCULAR_BUFFER;
	init : BOOL;
	id : WORD;
END_VAR

(*
version 1.0		01. jan. 2011
programmer		ks
tested by			ks

DLOG_DT legt den formatierten DT String im FIFO-RING-Buffer ab um diesen mit den Baustein DLOG_STORE_*  aufzuzeichnen
*)
IF NOT init THEN
	init := TRUE;
	X.ID_MAX := X.ID_MAX + 1;
	id := SHL(USINT_TO_WORD(X.ID_MAX),8) OR 1;
END_IF;

IF X.ADD_HEADER THEN
	X.UCB.D_STRING := COLUMN;
ELSIF X.ADD_DATA THEN
	X.UCB.D_STRING := DT_TO_STRF(DTI:=X.DTI,MS:=0,FMT:=FMT,LANG:=0);
ELSE
	RETURN;
END_IF;
X.UCB.D_HEAD := id;
X.UCB.D_MODE := 1;
UCB(DATA:=X.UCB); (* Daten eintragen *)
END_FUNCTION_BLOCK

(* POU DLOG_REAL, ST *)
FUNCTION_BLOCK DLOG_REAL
VAR_IN_OUT
	X : DLOG_DATA;
END_VAR
VAR_INPUT
	VALUE : REAL;
	N : INT;
	COLUMN : STRING;
END_VAR
VAR
	UCB : UNI_CIRCULAR_BUFFER;
	init : BOOL;
	id : WORD;
END_VAR

(*
version 1.0		01. jan. 2011
programmer		ks
tested by			ks

DLOG_REAL legt den REAL-Wert als STRING im FIFO-RING-Buffer ab um diesen mit den Baustein DLOG_STORE_*  aufzuzeichnen
*)
IF NOT init THEN
	init := TRUE;
	X.ID_MAX := X.ID_MAX + 1;
	id := SHL(USINT_TO_WORD(X.ID_MAX),8) OR 1;
END_IF;

IF X.ADD_HEADER THEN
	X.UCB.D_STRING := COLUMN;
ELSIF X.ADD_DATA THEN
	X.UCB.D_STRING := REAL_TO_STRF(IN:=VALUE,N:=N);
ELSE
	RETURN;
END_IF;
X.UCB.D_HEAD := id;
X.UCB.D_MODE := 1;
UCB(DATA:=X.UCB); (* Daten eintragen *)

(* revision history
ks	01. jan. 2011	rev 1.0
	original version
*)
END_FUNCTION_BLOCK

(* POU DLOG_DINT, ST *)
FUNCTION_BLOCK DLOG_DINT
VAR_IN_OUT
	X : DLOG_DATA;
END_VAR
VAR_INPUT
	VALUE : DINT;
	COLUMN : STRING;
END_VAR
VAR
	UCB : UNI_CIRCULAR_BUFFER;
	init : BOOL;
	id : WORD;
END_VAR

(*
version 1.0		01. jan. 2011
programmer		ks
tested by			ks

DLOG_DINT legt den DINT-Wert als STRING im FIFO-RING-Buffer ab um diesen mit den Baustein DLOG_STORE_* aufzuzeichnen
*)
IF NOT init THEN
	init := TRUE;
	X.ID_MAX := X.ID_MAX + 1;
	id := SHL(USINT_TO_WORD(X.ID_MAX),8) OR 1;
END_IF;

IF X.ADD_HEADER THEN
	X.UCB.D_STRING := COLUMN;
ELSIF X.ADD_DATA THEN
	X.UCB.D_STRING := DINT_TO_STRING(VALUE);
ELSE
	RETURN;
END_IF;
X.UCB.D_HEAD := id;
X.UCB.D_MODE := 1;
UCB(DATA:=X.UCB); (* Daten eintragen *)

(* revision history
ks	01. jan. 2011	rev 1.0
	original version
*)
END_FUNCTION_BLOCK

(* POU DLOG_FILE_TO_FTP, ST *)
FUNCTION_BLOCK DLOG_FILE_TO_FTP
VAR_IN_OUT
	X : DLOG_DATA;
END_VAR
VAR_INPUT
	FTP_URL : STRING(STRING_LENGTH);
	FTP_ACTIV : BOOL;
	FILE_DELETE : BOOL;
	TIMEOUT : TIME := T#30s;
	RETRY : INT;
	RETRY_TIME : TIME := T#30s;
	DNS_IP4 : DWORD;
	PLC_IP4 : DWORD;
END_VAR
VAR_OUTPUT
	DONE : BOOL;
	BUSY : BOOL;
	ERROR_C : DWORD;
	ERROR_T : BYTE;
END_VAR
VAR
	UCBD : UNI_CIRCULAR_BUFFER_DATA;
	UCB : UNI_CIRCULAR_BUFFER;
	FTP_CLIENT : FTP_CLIENT;
	WT_1 : TON;
	ftrig_old : BOOL;
	filename : STRING;
	step : INT;
	ftp_busy : BOOL;
	ftp_done : BOOL;
	cnt : INT;

	(*FB_LOG_MESSAGE : LOG_MSG;
	_debug_enable : BOOL := TRUE;*)
END_VAR

(*
version 1.0		01. jan. 2011
programmer		ks
tested by			ks

DLOG_FILE_TO_FTP der Baustein kopiert bzw verschiebt die vom DLOG_STORE_FILE_CSV erzeugten Dateien auf einem FTP-Server
*)
(* neue Filenamen speichern *)
IF X.NEW_FILE_RTRIG AND ftrig_old = FALSE THEN
	UCBD.D_HEAD := 1;
	UCBD.D_MODE := 1;
	UCBD.D_STRING := X.NEW_FILE;
	UCB(DATA:=UCBD); (* Daten eintragen *)
END_IF;
ftrig_old := X.NEW_FILE_RTRIG;

CASE step OF

00:	IF UCBD.BUF_COUNT > 0 AND ftp_busy = FALSE THEN
		UCBD.D_MODE := 10; (* Daten lesen *)
		UCB(DATA:=UCBD);
		UCBD.D_MODE := 11; (* Daten löschen *)
		UCB(DATA:=UCBD);
		filename := UCBD.D_STRING;
		cnt := 0;
		step := 10;
	END_IF;

10:	IF ftp_busy = FALSE THEN
		IF ftp_done THEN
			(*####################  DEBUG-MESSAGE  ###################################*)
			(*IF _debug_enable THEN
				LOG_CL.NEW_MSG := 'F_T_FTP: /FILE OK >~1<';
				LOG_CL.PRINTF[1] := filename;
				FB_LOG_MESSAGE();
			END_IF;*)
			(*########################################################################*)
			step := 0;
		ELSE
			step := 20; (* pause nach error *)
		END_IF;
	END_IF;

20:	IF WT_1.Q THEN (* Wartezeit *)
		cnt := cnt - 1;
		IF RETRY = 0 THEN (* FTP Transfer unbegrenzt wiederholen *)
			(*####################  DEBUG-MESSAGE  ###################################*)
			(*IF _debug_enable THEN
				LOG_CL.NEW_MSG := 'F_T_FTP: Auftrag unbegrenzt wiederholen /file: ~2';
				LOG_CL.PRINTF[2] := filename;
				FB_LOG_MESSAGE();
			END_IF;*)
			(*########################################################################*)
			step := 10; (* FTP Transfer wiederholen *)
		ELSIF cnt >= 0 THEN
			(*####################  DEBUG-MESSAGE  ###################################*)
			(*IF _debug_enable THEN
				LOG_CL.NEW_MSG := 'F_T_FTP: Auftrag wiederholen /cnt: ~1 /file: ~2';
				LOG_CL.PRINTF[1] := INT_TO_STRING(cnt);
				LOG_CL.PRINTF[2] := filename;
				FB_LOG_MESSAGE();
			END_IF;*)
			(*########################################################################*)
			step := 10; (* FTP Transfer wiederholen *)
		ELSE
			(*####################  DEBUG-MESSAGE  ###################################*)
			(*IF _debug_enable THEN
				LOG_CL.NEW_MSG := 'F_T_FTP: Auftrag verworfen /file: ~2';
				LOG_CL.PRINTF[2] := filename;
				FB_LOG_MESSAGE();
			END_IF;*)
			(*########################################################################*)
			step := 0; (* FTP Auftrag verwerfen *)
		END_IF;
	END_IF;

END_CASE;

BUSY := step = 10;
DONE := step = 0;
WT_1(IN:= step = 20, PT:= RETRY_TIME);

FTP_CLIENT(
	ACTIVATE:= BUSY,
	FILENAME:= filename,
	FTP_URL:= FTP_URL,
	FTP_DOWNLOAD:= FALSE,
	FTP_ACTIV:= FTP_ACTIV,
	FILE_DELETE:= FILE_DELETE,
	TIMEOUT:= TIMEOUT,
	DNS_IP4:= DNS_IP4,
	PLC_IP4:= PLC_IP4,
	DONE=> ftp_done,
	BUSY=> ftp_busy,
	ERROR_C=> ERROR_C,
	ERROR_T=> ERROR_T
	);

(* revision history
ks	01. jan. 2011	rev 1.0
	original version
*)
END_FUNCTION_BLOCK

(* POU FTP_CLIENT, ST *)
(* @OBJECTFLAGS := '0, 8' *)
FUNCTION_BLOCK FTP_CLIENT
VAR_INPUT
	ACTIVATE : BOOL;
	FILENAME : STRING;
	FTP_URL : STRING(STRING_LENGTH);
	FTP_DOWNLOAD : BOOL;
	FTP_ACTIV : BOOL;
	FILE_DELETE : BOOL;
	TIMEOUT : TIME;
	DNS_IP4 : DWORD;
	PLC_IP4 : DWORD;
END_VAR
VAR_OUTPUT
	DONE : BOOL;
	BUSY : BOOL;
	ERROR_C : DWORD;
	ERROR_T : BYTE;
END_VAR
VAR
	IP_C1 : IP_C; (* IP_Control Verwaltungsstruktur *)
	IP_C2 : IP_C; (* IP_Control Verwaltungsstruktur *)
	S_BUF1 : NETWORK_BUFFER;
	S_BUF2 : NETWORK_BUFFER;
	R_BUF1 : NETWORK_BUFFER;
	R_BUF2 : NETWORK_BUFFER;
	URL_DATA : url;
	DNS_CLIENT : DNS_CLIENT;
	IPC1 : IP_CONTROL;
	IPC2 : IP_CONTROL;
	FS : FILE_SERVER;
	FSD : FILE_SERVER_DATA;

	activate_last : BOOL;
	step : INT;
	snd_step : INT;
	snd_text :	STRING(STRING_LENGTH);
	rcv_text :	STRING(STRING_LENGTH);
	rcv_state : INT;
	TON_WAIT : TON;
	last_step : INT;
	next_step : INT;
	idx1 : INT;
	idx2 : INT;
	str1 : STRING(STRING_LENGTH);
	str2 : STRING(STRING_LENGTH);
	ftp_path : STRING;
	byar : ARRAY [0..5] OF BYTE;
	dw_tmp : DWORD;
	w_tmp : WORD;
	fpd : FILE_PATH_DATA;
	timeout2 : TIME;
	ftp_file_size : UDINT;

	(*FB_LOG_MESSAGE : LOG_MSG;
	_debug_enable : BOOL := FALSE;*)

END_VAR
(*
version 1.1		06.apr. 2011
programmer		ks
tested by			ks

FTP_CLIENT dient zum senden und empfangen von dateien von einem FTP-Server.



110 Restart marker reply 										Markierung für Wiederaufnahme der Übertragung 
120 Service ready in x minutes 									Dienst steht in x Minuten zu Verfügung 
125 Data connection already open; 								transfer starting Datenverbindung besteht bereits; beginne mit der Übertragung 
150 File status okay; about to open data connection 					Dateistatus OK; Datenverbindung wird aufgebaut 
200 Command okay 											Befehl OK 
202 Command not implemented 									Befehl nicht implementiert 
211   														Antwort für Systemstatus oder Hilfefunktion des Systems 
212   														Verzeichnisstatus 
213   														Dateistatus 
214   														Meldung der Hilfefunktion 
215 NAME system type 										Angabe des Systemtyps 
220 Service ready for new user 									Dienst bereit für neuen Benutzer 
221 Service closing control connection 							Steuerverbindung des Dienstes wird getrennt; Benutzer wird abgemeldet 
225 Data connection open; no transfer in progress 					Datenverbindung hergestellt; derzeit keine Übertragung 
226 Closing data connection. Requested file action successful 		Datenverbindung wird getrennt 
227 Entering Passive Mode 										Passiver Modus aktiviert 
230 User logged in, proceed 									Benutzer angemeldet, bitte fortfahren 
250 Requested file action okay, completed 						Angeforderter Vorgang OK, beendet 
257 "PATH" created 											"PFAD" wurde erstellt 
331 User name okay, need password 							Benutzername OK, Kennwort erforderlich 
332 Need account for login 										Benutzerkonto zur Anmeldung erforderlich 
350 Requested file action pending further information 				Mehr Informationen für Dateivorgang erforderlich 
421 Service not available, closing control connection 				Dienst nicht verfügbar, Steuerverbindung wird getrennt 
425 Can't open data connection 									Datenverbindung kann nicht hergestellt werden 
426 Connection closed; transfer aborted Verbindung getrennt; 		Übertragung abgebrochen 
450 Requested file action not taken; File unavailable 				Angeforderter Dateivorgang wurde nicht ausgeführt; Datei nicht verfügbar 
451 Requested action aborted: local error in processing 				Angeforderter Vorgang abgebrochen: Lokaler Fehler bei der Bearbeitung 
452 Requested action not taken; Insufficient storage space in system 	Angeforderter Vorgang nicht ausgeführt; Nicht genügend Speicherplatz auf System 
500 Syntax error 												Befehl nicht erkannt 
501 Syntax error in parameters or arguments 						Syntaxfehler bei den Parametern 
502 Command not implemented 									Befehl nicht implementiert 
503 Bad sequence of commands 								Ungültige Befehlsabfolge 
504 Command not implemented for that parameter 					Befehl für diesen Parameter nicht implementiert 
530 Not logged in 												Nicht angemeldet 
532 Need account for storing files 								Zum Speichern von Dateien Anmeldung erforderlich 
550 Requested file action not taken; File unavailable Angeforderter 	Dateivorgang wurde nicht ausgeführt; Datei nicht verfügbar 
551 Requested action aborted: page type unknown 					Angeforderter Vorgang abgebrochen: Unbekannter Seitentyp 
552 Requested file action aborted: Exceeded storage allocation 		Angeforderter Dateivorgang abgebrochen: Nicht genügend Platz in aktuellem Verzeichnis oder Datensatz 
553 Requested action not taken: File name not allowed 				Angeforderter Vorgang nicht ausgeführt: Unzulässiger Dateiname 

#########################
ERROR_T

1 = DNS_CLIENT
2 = FTP Steuerkanal
3 = FTP Datenkanal
4 = FILE_SERVER
5 = Ablaufstörung
#########################

*)
CASE step OF

00:	IF ACTIVATE AND NOT activate_last THEN
		ftp_file_size := UDINT#0;
		timeout2 := TIMEOUT + T#1s;
		DONE := FALSE;
		ERROR_C := DWORD#0;
		ERROR_T := BYTE#0;
		FSD.ERROR := BYTE#0;
		URL_DATA := STRING_TO_URL(STR:=FTP_URL,DEFAULT_PROTOCOL:='',DEFAULT_PATH:='/');
		IF LEN(URL_DATA.USER) = 0 THEN
			URL_DATA.USER := 'Anonymous';
			URL_DATA.PASSWORD := 'User@';
		END_IF;

		FILE_PATH_SPLIT(FILENAME:=FILENAME,X:=fpd); (* Datei-Path zerlegen *)
		str1 := fpd.FILENAME; (* zwischenspeichern *)
		FILE_PATH_SPLIT(FILENAME:=URL_DATA.PATH,X:=fpd); (* FTP-Path zerlegen *)
		IF LEN(fpd.FILENAME) = 0 THEN (* wenn FTP-Path keinen Dateinamen enthält , dann den Namen der lokalen Datei benutzen *)
			ftp_path := CONCAT(URL_DATA.PATH,str1);
		ELSE
			ftp_path := URL_DATA.PATH;
		END_IF;
		step := 10;
	END_IF;

10:	IF DNS_CLIENT.DONE THEN
		step := 20;
	ELSIF DNS_CLIENT.ERROR <> DWORD#0 THEN
		ERROR_C := DNS_CLIENT.ERROR;
		ERROR_T := BYTE#1;
		step := 980;
	END_IF;

20:	(* FTP Steuerkanal einrichten *)
	IP_C1.C_PORT := WORD#21; (* Portnummer eintragen *)
  	IP_C1.C_IP := DNS_CLIENT.IP4; (* IP eintragen *)
  	IP_C1.C_MODE := BYTE#0; (* Mode: TCP+ACTIV+PORT *)
  	IP_C1.TIME_RESET := TRUE; (* Zeitueberwachung rücksetzen *)
  	IP_C1.C_ENABLE := TRUE; (* Verbindungsaufbau freigeben *)
  	IP_C1.R_OBSERVE := TRUE; (* Empfangsueberwachung *)
	R_BUF1.SIZE := UINT#0;

  	IP_C2.C_ENABLE   := FALSE; (* Verbindungsaufbau sperren *)
	step := 30;

30:	IF rcv_state = 220 THEN (* 220 = Service ready for new user *)
		snd_text := CONCAT('USER ',URL_DATA.USER);
		next_step := 40;
	END_IF;

40:	IF rcv_state = 331 THEN (* 331 = User name okay, need password *)
		snd_text := CONCAT('PASS ',URL_DATA.PASSWORD);
		next_step := 50;
	ELSIF rcv_state = 230 THEN (* 230 = User logged in, proceed *)
		next_step := 50;
	ELSIF rcv_state = 220 THEN (* 220 = Service ready for new user *)
		next_step := 20; (* WORK verbindung sollte ab/aufgebaut werden *)
	END_IF;

50:	IF rcv_state = 230 THEN (* 230 = User logged in, proceed *)
		snd_text := 'TYPE I';  (* binären Modus aktivieren *)
		next_step := 54;
	END_IF;

54:	IF rcv_state = 200 THEN (* 200 = Command okay *)
		IF FTP_DOWNLOAD THEN (* Datei von FTP Empfangen *)
			snd_text := CONCAT('SIZE ', ftp_path); (* SIZE /PFAD/FILENAME *)
			next_step := 56;
		ELSE
			step := 60;
		END_IF;
	END_IF;

56:	IF rcv_state = 213 THEN (* 213 Filesize *)
		str1 := ELEMENT_GET(SEP:=BYTE#32,POS:=1,ELEMENT:=rcv_text);
		ftp_file_size := STRING_TO_UDINT(str1); (* Dateigroesse in bytes gestimmen *)
		step := 60;
	END_IF;

60:	IF FTP_ACTIV THEN (* FTP Server aktiv *)
		IF URL_DATA.PORT = WORD#0 THEN
			URL_DATA.PORT := WORD#20; (* Standard Datenkanal *)
		END_IF;
		str2 := '';
		dw_tmp := PLC_IP4;
		FOR idx1 := 0 TO 5 DO
			IF idx1 = 4 THEN
				dw_tmp := ROR(WORD_TO_DWORD(URL_DATA.PORT),8);
			ELSE
				dw_tmp := ROL(dw_tmp,8);
			END_IF;
			str2 := CONCAT(str2,BYTE_TO_STRING(DWORD_TO_BYTE(dw_tmp)));
			IF idx1 < 5 THEN
				str2 := CONCAT(str2,',');
			END_IF;
		END_FOR;
		dw_tmp := DNS_CLIENT.IP4; (* IP eintragen *)
		w_tmp := URL_DATA.PORT; (* Port Nummer des Datenkanals *)
		snd_text := CONCAT('PORT ',str2); (* FTP Server in den aktiv-mode schalten *)
		next_step := 80;
	ELSE
		snd_text := 'PASV';  (* FTP Server in den passiv-mode schalten *)
		next_step := 70;
	END_IF;
	step := 999; (* Warten auf next_step *)

70:	IF rcv_state = 227 THEN (* 227 = Entered Passive Mode (213,202,225,43,212,186) *)
		idx1 := FIND(rcv_text , '(' );
		idx2 := FIND(rcv_text , ')' );
		IF idx1 > 0 AND idx2 > idx1+1 THEN
			str1 := MID(rcv_text, idx2 - idx1 - 1, idx1+1);
			FOR idx1 := 0 TO 5 DO
				str2 := ELEMENT_GET(SEP:=BYTE#44,POS:=idx1,ELEMENT:=str1);
				byar[idx1] := STRING_TO_BYTE(str2);
			END_FOR;
			dw_tmp := DWORD_OF_BYTE(byar[0],byar[1],byar[2],byar[3]); (* IP Adresse des Datenkanals *)
			w_tmp := WORD_OF_BYTE(byar[4],byar[5]); (* Port Nummer des Datenkanals *)
		END_IF;
		step := 100;
	END_IF;

80:	IF rcv_state = 200 THEN (* 200 = PORT command successful *)
		step := 100;
	END_IF;

100:IP_C2.C_MODE := SEL(FTP_ACTIV,BYTE#0,BYTE#2); (* Aktiv = Mode 2: TCP+PASSIV+PORT / passiv = Mode 0: TCP+ACTIV+PORT *)
	IP_C2.C_IP := dw_tmp; (* IP Adresse des Datenkanals *)
	IP_C2.C_PORT := w_tmp; (* Port Nummer des Datenkanals *)
  	IP_C2.TIME_RESET := TRUE; (* Zeitueberwachung rücksetzen *)
  	IP_C2.C_ENABLE := TRUE; (* Verbindungsaufbau freigeben *)
	IP_C2.R_OBSERVE := FALSE; (* Empfangsueberwachung *)
	R_BUF2.SIZE := UINT#0;
	step := 120;

120:IF IP_C2.C_STATE > BYTE#127 THEN (* FTP Datenkanal aufgebaut *)
		IF FTP_DOWNLOAD THEN (* File von FTP empfangen *)
			IP_C2.MAILBOX[3] := BYTE#1; (* IP Empfang sperren *)
			step := 400;
		ELSE
			snd_text := 'STOR ';
			next_step := 140;
			snd_text := CONCAT(snd_text, ftp_path); (* STORE /PFAD/FILENAME *)
			step := 999; (* Warten auf next_step *)
		END_IF;
	END_IF;

(* ============== File an FTP senden ================ *)

140:IF rcv_state = 125 OR rcv_state = 150 THEN (* 125 = Data connection already open / 150 = File status okay; about to open data connection *)
		step := 160;
	END_IF;

160:FSD.FILENAME := FILENAME; (* Dateiname *)
	FSD.MODE := BYTE#1; (* vorhandene Datei zum lesen öffnen *)
	FSD.OFFSET := UDINT#0; (* Start bei Dateianfang *)
	FSD.AUTO_CLOSE := T#0s; (* kein Auto-Close verwenden *)
	S_BUF2.SIZE := UINT#65535; (* maximale länge einlesen *)
	IP_C2.MAILBOX[2] := BYTE#1; (* IP Senden blockieren *)
	step := 200;

200:IF FSD.MODE = BYTE#0 AND FSD.ERROR = BYTE#0 THEN
		IP_C2.MAILBOX[2] := BYTE#0; (* IP Senden erlauben *)
		step := 210;
	END_IF;

210:IF S_BUF2.SIZE = UINT#0 THEN (* warten bis alle daten gesendet sind *)
		IF FSD.FILE_SIZE - FSD.OFFSET > UDINT#0 THEN
			FSD.MODE := BYTE#1; (* vorhandene Datei zum lesen öffnen *)
			S_BUF2.SIZE := UINT#65535; (* maximale länge einlesen *)
			IP_C2.MAILBOX[2] := BYTE#1; (* IP Senden blockieren *)
			step := 200;
		ELSE
			IP_C2.C_ENABLE := FALSE; (* FTP Datenkanal schliessen *)
			step := 300;
		END_IF;
	END_IF;

300:IF rcv_state = 226 THEN (* 226 Closing data connection. Requested file action successful  *)
		snd_text := 'QUIT';
		next_step := 320;
	END_IF;

320:IF rcv_state = 221 THEN (* 221 Service closing control connection  *)
		IP_C1.C_ENABLE := FALSE; (* FTP Steuerkanal schliessen *)
		IF FILE_DELETE THEN (* Datei nach transfer löschen *)
			FSD.MODE := BYTE#4; (* File Remove *)
			step := 340;
		ELSE
			step := 900;
		END_IF;
	END_IF;

340:IF FSD.MODE = BYTE#0 AND FSD.ERROR = BYTE#0 THEN
		step := 900;
	END_IF;

(*  ============== File vom FTP Empfangen  ============== *)

400:snd_text := 'RETR ';
	next_step := 410;
	snd_text := CONCAT(snd_text, ftp_path); (* RETR /PFAD/FILENAME *)
	step := 999; (* Warten auf next_step *)

410:IF rcv_state = 125 OR rcv_state = 150 THEN (* 125 = Data connection already open / 150 = File status okay; about to open data connection *)
		IP_C2.R_OBSERVE := TRUE; (* Empfangsueberwachung *)
		step := 420;
	END_IF;

420:FSD.FILENAME := FILENAME; (* Dateiname *)
	FSD.MODE := BYTE#3; (* Datei neu anlegen *)
	FSD.OFFSET := UDINT#0; (* Start bei Dateianfang *)
	FSD.AUTO_CLOSE := T#0s; (* kein Auto-Close verwenden *)
	step := 460;

440:IF R_BUF2.SIZE > UINT#0 THEN (* warten bis daten empfangen wurden *)
		IP_C2.MAILBOX[3] := BYTE#1; (* IP Empfang blockieren bis Daten in Datei geschrieben wurden *)
		FSD.MODE := BYTE#3; (* Daten in Datei schreiben *)
		step := 460;
	ELSIF FSD.FILE_SIZE = ftp_file_size THEN (* Verbindung abgebaut ? , oder 226 = Closing data connection. Requested file action successful *)
		IP_C2.C_ENABLE := FALSE; (* FTP Datenkanal schliessen *)
		step := 700;
	END_IF;

460:IF FSD.MODE = BYTE#0 AND FSD.ERROR = BYTE#0 THEN (* warten bis Daten geschreiben wurden *)
		R_BUF2.SIZE := UINT#0; (* Daten löschen *)
		IP_C2.MAILBOX[3] := BYTE#0; (* IP Empfang wieder erlauben *)
		step := 440;
	END_IF;

(* ================================================== *)

700:IF rcv_state = 226 OR IP_C2.C_STATE < BYTE#127 THEN (* 226 Closing control connection. Requested file action successful  *)
		IF FTP_DOWNLOAD AND FILE_DELETE THEN (* FTP Download und File löschen ? *)
			snd_text := CONCAT('DELE ', ftp_path); (* DELE /PFAD/FILENAME *)
			next_step := 720;
		ELSE
			step := 740;
		END_IF;
	END_IF;

720:IF rcv_state = 250 THEN (* 250 Requested file action okay, completed *)
		step := 740;
	END_IF;

740:snd_text := 'QUIT';
	next_step := 760;
	step := 999; (* Warten auf next_step *)

760:IF rcv_state = 221 THEN (* 221 Service closing control connection  *)
		IP_C1.C_ENABLE := FALSE; (* FTP Steuerkanal schliessen *)
		IF NOT FTP_DOWNLOAD AND FILE_DELETE THEN (* FTP Upload und Datei nach transfer löschen *)
			FSD.MODE := BYTE#4; (* File Remove *)
			step := 780;
		ELSE
			step := 900;
		END_IF;
	END_IF;

780:IF FSD.MODE = BYTE#0 AND FSD.ERROR = BYTE#0 THEN
		step := 900;
	END_IF;

(* ================================================== *)

900:DONE := TRUE;
	step := 980;

980:IP_C1.C_ENABLE := FALSE; (* FTP Steuerkanal schliessen *)
	IP_C2.C_ENABLE := FALSE; (* FTP Datenkanal schliessen *)
	IP_C2.MAILBOX[2] := BYTE#0; (* IP Senden wieder erlauben *)
	IP_C2.MAILBOX[3] := BYTE#0; (* IP Empfang wieder erlauben *)
	S_BUF1.SIZE := UINT#0;
	S_BUF2.SIZE := UINT#0;
	R_BUF1.SIZE := UINT#0;
	R_BUF2.SIZE := UINT#0;
	ftp_file_size := UDINT#0;
	snd_step := 0;
	next_step := 0;
	FSD.MODE := BYTE#5; (* Datei schliessen *)
	step := 990;

990:IF IP_C1.C_STATE = BYTE#0 AND IP_C2.C_STATE = BYTE#0 AND FSD.FILE_OPEN = FALSE THEN
		step := 0;
	END_IF;

999: ; (* Dummy Schritt, warten bis neuer schritt durch "next_step" aktiv wird *)

END_CASE;

(* ++++++++++++++++++++++++++++++++++++++++++++++++++++++++++ *)

IF step >= 30 THEN
	IF R_BUF1.SIZE > UINT#0 THEN (* Daten wurden empfangen ? *)
		idx1 := UINT_TO_INT(R_BUF1.SIZE);
		REPEAT (* zeilenterminierung erkennen und echtes TEXT-Ende bestimmen *)
			idx1 := idx1 - 1;
		UNTIL idx1 = 0 OR R_BUF1.BUFFER[idx1] >= BYTE#32 (* TRUE = EXIT *)
		END_REPEAT;
		idx1 := idx1 + 1; (* index auf SIZE umrechnen *)
		rcv_text := BUFFER_TO_STRING(PT:=ADR(R_BUF1.BUFFER),SIZE:=idx1,START:=0,STOP:=STRING_LENGTH-1);
		IF LEN(rcv_text) >= 3 THEN (* Statuscode prüfen und auswerten *)
			str1 := LEFT(rcv_text,3);
			IF IS_NUM(STR:=str1) THEN (* enthält nur Zahlen ? *)
				rcv_state := STRING_TO_INT(str1);
			END_IF;
			IP_C1.R_OBSERVE := FALSE;
		END_IF;
		R_BUF1.SIZE := UINT#0; (* daten löschen *)

	        (*####################  DEBUG-MESSAGE  ###################################*)
	        (*IF _debug_enable THEN
	          LOG_CL.NEW_MSG := 'RCV: >~1<';
	          LOG_CL.PRINTF[1] := rcv_text;
	          FB_LOG_MESSAGE();
	        END_IF;*)
	        (*########################################################################*)

	END_IF;
END_IF;

(* automatisches Datensenden *)

CASE snd_step OF

00:	IF LEN(snd_text) > 0 THEN
	        (*####################  DEBUG-MESSAGE  ###################################*)
	        (*IF _debug_enable THEN
	          LOG_CL.NEW_MSG := 'SND: >~1<';
	          LOG_CL.PRINTF[1] := snd_text;
	          FB_LOG_MESSAGE();
	        END_IF;*)
	        (*########################################################################*)
		_STRING_TO_BUFFER(str:=snd_text,pos:=0,pt:=ADR(S_BUF1.BUFFER),size:=SIZEOF(S_BUF1.BUFFER)); (* String in puffer kopieren *)
		idx1 := LEN(snd_text);
		S_BUF1.BUFFER[idx1] := BYTE#16#0D;
		idx1 := idx1 + 1;
		S_BUF1.BUFFER[idx1] := BYTE#16#0A;
		idx1 := idx1 + 1;
		S_BUF1.SIZE := INT_TO_UINT(idx1); (* Sendelänge eintragen *)
		R_BUF1.SIZE := UINT#0; (* Empfangsbuffer rücksetzen *)
		IP_C1.R_OBSERVE := TRUE;
		rcv_state := 9999; (* letzen FTP Status löschen *)
		snd_text := '';
		snd_step := 10;
	END_IF;

10:	IF S_BUF1.SIZE = UINT#0 THEN (* warten bis alle daten gesendet sind *)
		step := next_step;
		snd_step := 0;
	END_IF;

END_CASE;

(* Fehlerbehandlung *)
IF ERROR_T = BYTE#0 THEN (* noch kein Fehler gespeichert *)
	IF IP_C1.ERROR > DWORD#0 THEN (* IP Control 1 *)
		ERROR_C := IP_C1.ERROR;
		ERROR_T := BYTE#2;
		step := 980;
	ELSIF IP_C2.ERROR > DWORD#0 THEN (* IP Control 2 *)
		ERROR_C := IP_C2.ERROR;
		ERROR_T := BYTE#3;
		step := 980;
	ELSIF FSD.MODE = BYTE#0 THEN
		IF FSD.ERROR > BYTE#0 THEN
			ERROR_C := BYTE_TO_DWORD(FSD.ERROR);
			ERROR_T := BYTE#4; (* Dateizugriff *)
			step := 980;
		END_IF;
	END_IF;
END_IF;

IF TON_WAIT.Q THEN (* Ablaufstörung - Schrittkette *)
	ERROR_C := SHL(INT_TO_DWORD(step),16) OR INT_TO_DWORD(rcv_state); (* aktuellen Schritt und letzten FTP Status eintragen *)
	ERROR_T := BYTE#5;
	step := 980;
END_IF;

(* ######################################################## *)

DNS_CLIENT(IP_C:=IP_C1, S_BUF:=S_BUF1, R_BUF:=R_BUF1, DOMAIN:=URL_DATA.DOMAIN, IP4_DNS:= DNS_IP4, ACTIVATE:=step=10); (* DNS-Client *)
IPC1(IP:= DWORD#0, PORT:= WORD#0 , TIME_OUT:= TIMEOUT, IP_C:= IP_C1, S_BUF:= S_BUF1, R_BUF:= R_BUF1); (* FTP Steuerkanal *)
IPC2(IP:= DWORD#0, PORT:= WORD#0 , TIME_OUT:= TIMEOUT, IP_C:= IP_C2, S_BUF:= S_BUF2, R_BUF:= R_BUF2); (* FTP Datenkanal *)

TON_WAIT(IN:=step = last_step AND step > 0,PT:=timeout2);
last_step := step;
activate_last := ACTIVATE;
BUSY := step <> 0;

IF FTP_DOWNLOAD THEN (* FILE_SERVER *)
	FS(FSD:=FSD,PT:=R_BUF2); (* Datei von FTP empfangen *)
ELSE
	FS(FSD:=FSD,PT:=S_BUF2); (* Datei an FTP senden *)
END_IF;

(* revision history

ks	06. apr. 2011	rev 1.1
	list_len und list_get durch element_count und element_get ersetzt

ks	01. jan. 2011	rev 1.0
	original version
*)
END_FUNCTION_BLOCK

(* POU DNS_CLIENT, ST *)
FUNCTION_BLOCK DNS_CLIENT
VAR_IN_OUT
	IP_C : IP_C; (* IP_Control Verwaltungsstruktur *)
	S_BUF : NETWORK_BUFFER;
	R_BUF : NETWORK_BUFFER;
END_VAR
VAR_INPUT
	ACTIVATE : BOOL;
	DOMAIN : STRING;
	IP4_DNS : DWORD;
END_VAR
VAR_OUTPUT
	IP4 : DWORD;
	DONE : BOOL;
	ERROR : DWORD;
END_VAR
VAR
	IP_FIFO : IP_FIFO;
	ip_state : BYTE;
	ip_id : BYTE;
	i : INT;
	state : INT;
	domain_copy : STRING;
	activate_last : BOOL;
	url_length : INT;
	char : BYTE;
	char_count : INT;
	tid : BYTE;
	anc : INT;
	x : BYTE;
	rr_stop : BOOL;
	ttl_last : DWORD;
	ttl_tmp : DWORD;

END_VAR

(*
version 1.1	20. dec. 2010
programmer 	ks
tested BY	ks

DNS_CLIENT führt eine Domain-Name Abfrage bei einen DNS-Server durch

*)
(* Domain Name System (query) *)

CASE state OF

00:	IF ACTIVATE AND NOT activate_last THEN (* auf positive Flanke GET warten *)
		DONE := FALSE;
		ERROR := DWORD#0;
		state := 5;
	END_IF;

05:	IP4 := IP4_DECODE(str:=DOMAIN); (* prüfe ob domain schon eine IP4-Adresse ist *)
	IF IP4 > DWORD#00 THEN
		DONE := TRUE;
		state := 0;
	ELSE
		ip_state := BYTE#1;
		ttl_last := DWORD#0;
		domain_copy := DOMAIN; (* DOMAIN String sichern *)
		state := 10;
	END_IF;

10:	IF ip_state = BYTE#3 THEN (* Bei IP_Control anmelden *)
		url_length := LEN(domain_copy);
		char_count := 17 + url_length; (* sendebuffer initialisieren *)
		FOR i := 0 TO char_count DO
			S_BUF.BUFFER[i] := BYTE#00;
		END_FOR;
		tid := UINT_TO_BYTE(BYTE_TO_UINT(tid) + UINT#1);
		S_BUF.BUFFER[01] := tid; (* Transaction ID lowbyte *)
		S_BUF.BUFFER[02] := BYTE#16#01; (* Flags: highbyte *)
		S_BUF.BUFFER[05] := BYTE#16#01; (* Questions: lowbyte *)
		i := url_length + 12;	(* den servernamen von hinten nach vorne bearbeiten *)
		char_count := 0;
		WHILE i > 12 DO
			char := CODE(STR:=domain_copy,POS:=i - 12);
			IF char = BYTE#46 THEN (* prüfe auf haupt/sub domänen namens-teiler "." *)
				S_BUF.BUFFER[i] := INT_TO_BYTE(char_count); (* anstelle des teilers "." wird die länge des erkannten haupt/sub domänennames eingetragen *)
				char_count := 0;
			ELSE
				S_BUF.BUFFER[i] := char; (* char in buffer eintragen *)
				char_count := char_count + 1; (* anzahl char zählen *)
			END_IF;
			i := i - 1;
		END_WHILE;
		S_BUF.BUFFER[i] := INT_TO_BYTE(char_count); (* längenangabe des ganz linken (ersten) domänennamens eintragen *)
		i := url_length + 15; (* position hinter dem servernamen *)
		S_BUF.BUFFER[i] := BYTE#01; (* Type: A Hostaddress lowbyte *)
		i := i + 2;
		S_BUF.BUFFER[i] := BYTE#01; (* Class: IN lowbyte *)
		i := i + 1;
		(* IP Datenverkehr einrichten *)
		IP_C.C_PORT := WORD#53; (* Portnummer eintragen *)
		IP_C.C_IP := IP4_DNS; (* IP eintragen *)
		IP_C.C_MODE := BYTE#1; (* Mode: UDP+AKTIV+PORT+IP *)
		IP_C.C_ENABLE := TRUE; (* Verbindungsaufbau freigeben *)
		IP_C.TIME_RESET := TRUE; (* Zeitueberwachung rücksetzen *)
		IP_C.R_OBSERVE  := TRUE; (* Datenempfang ueberwachen *)
		S_BUF.SIZE := INT_TO_UINT(i); (* sendelänge eintragen *)
		R_BUF.SIZE := UINT#0; (* Empfangslänge rücksetzen *)
		state := 30;
	END_IF;

30:	IF IP_C.ERROR <> DWORD#00 THEN
		ERROR := IP_C.ERROR;
		state := 99;
	ELSIF (S_BUF.SIZE = UINT#0) AND (tid = R_BUF.BUFFER[1]) AND (R_BUF.SIZE >= INT_TO_UINT(34 + url_length)) THEN	(* prüfe ob antwort telegramm die richtige Transaction-ID und mindestlänge hat *)
		ERROR := BYTE_TO_DWORD(R_BUF.BUFFER[3] AND BYTE#2#0000_1111); (* prüfe Return code der Flags. 4 bits *)
		IF ERROR = DWORD#00 THEN
			anc := R_BUF.BUFFER[7]; (* Anzahl der Answer-RR *)
			IP_C.R_OBSERVE := FALSE; (* Datenempfang ueberwachen *)
			state := 40;
		ELSE
			state := 99;
		END_IF;
	END_IF;

40:	IF anc > 0 THEN
		anc := anc - 1;
		WHILE i < R_BUF.SIZE DO
			x := R_BUF.BUFFER[i];
			IF rr_stop = FALSE THEN
				IF x > BYTE#63 THEN (* zeiger auf namen *)
					i := i + 1;
					rr_stop := TRUE;
				ELSIF x= BYTE#0 THEN (* namens ende *)
					rr_stop := TRUE;
				ELSE
					i := i + x; (* namen *)
				END_IF;
				i := i + 1;
			ELSE
				rr_stop := FALSE;
				IF R_BUF.BUFFER[i+1] = BYTE#1 AND R_BUF.BUFFER[i+3] = BYTE#1 THEN (* Type A / Class IN *)
					i := i + 4;
					ttl_tmp := DWORD_OF_BYTE(R_BUF.BUFFER[i],R_BUF.BUFFER[i+1],R_BUF.BUFFER[i+2],R_BUF.BUFFER[i+3]); (* Time to live *)
					i := i + 6;
					IF ttl_tmp >= ttl_last THEN (* TTL ist länger *)
						ttl_last := ttl_tmp;
						IP4 := DWORD_OF_BYTE(R_BUF.BUFFER[i],R_BUF.BUFFER[i+1],R_BUF.BUFFER[i+2],R_BUF.BUFFER[i+3]); (* IP-Adresse *)
					END_IF;
					i := i + 4;
				ELSE
					i := i + 9;
					i := i + R_BUF.BUFFER[i] + 1; (* offset zu nächsten Block *)
				END_IF;
				EXIT;
			END_IF;
		END_WHILE;
	ELSE
		IF ttl_last > DWORD#0 THEN (* gültige RR mit IP gefunden *)
			DONE := TRUE;
		END_IF;
		state := 99;
	END_IF;

99:	R_BUF.SIZE := UINT#0; (* Empfangslänge rücksetzen *)
	ip_state := BYTE#4; (* Abmelden *)
	state := 00;

END_CASE;

activate_last := ACTIVATE; (* letzten Status sichern zur Flankenerkennung *)
IP_FIFO(FIFO:=IP_C.FIFO,STATE:=ip_state,ID:=ip_id); (* IP_FIFO *)

(* revision history

ks	18. oct. 2008	rev 1.0
	original version

ks	20. oct. 2009	rev 1.1
	unbenutzten code entfernt, all buffer base 0

ks	20. dec. 2010	rev 1.2
	parsing nach rfc1305
*)


(*----------------------------------------------------------------------------------------------------------------*)
(* Flags: 0x0100 (Standard query)                                                                                            *)
(* 0... .... .... .... = Response: Message is a query                                                                   *)
(* .000 0... ....  = Opcode: Standard query (0)                                                                          *)
(* .... ..0. .... .... = Truncated: Message is not truncated                                                          *)
(* .... ...1 .... .... = Recursion desired: Do query recursively                                                    *)
(* .... .... .0.. .... = Z: reserved (0)                                                                                                  *)
(* .... .... ...0 .... = Non-authenticated data OK: Non-authenticated data is unacceptable *)
(*-----------------------------------------------------------------------------------------------------------------*)

(*      0  1  2  3  4  5  6  7  8  9  0  1  2  3  4  5  *)
(*    +--+--+--+--+--+--+--+--+--+--+--+--+--+--+--+--+ *)
(*    |                      ID                       | idx: 0/1   *)
(*    +--+--+--+--+--+--+--+--+--+--+--+--+--+--+--+--+ *)
(*    |QR|   Opcode  |AA|TC|RD|RA|   Z    |   RCODE   | idx: 2/3   *)
(*    +--+--+--+--+--+--+--+--+--+--+--+--+--+--+--+--+ *)
(*    |                    QDCOUNT                    | idx: 4/5   *)
(*    +--+--+--+--+--+--+--+--+--+--+--+--+--+--+--+--+ *)
(*    |                    ANCOUNT                    | idx: 6/7   *)
(*    +--+--+--+--+--+--+--+--+--+--+--+--+--+--+--+--+ *)
(*    |                    NSCOUNT                    | idx: 8/9   *)
(*    +--+--+--+--+--+--+--+--+--+--+--+--+--+--+--+--+ *)
(*    |                    ARCOUNT                    | idx: 10/11 *)
(*    +--+--+--+--+--+--+--+--+--+--+--+--+--+--+--+--+ *)

